LIN {X 0.182,Y -641.756,Z 1201.615,A 0.000,B 0.000,C 90.000,E1 146.755} C_DIS
LIN {X 0.071,Y -644.719,Z 1201.609,A 0.000,B 0.000,C 90.000,E1 145.515} C_DIS
LIN {X -0.049,Y -646.870,Z 1201.603,A 0.000,B 0.000,C 90.000,E1 144.529} C_DIS
LIN {X -0.142,Y -649.015,Z 1201.597,A 0.000,B 0.000,C 90.000,E1 143.543} C_DIS
LIN {X -0.312,Y -652.420,Z 1201.588,A 0.000,B 0.000,C 90.000,E1 141.823} C_DIS
LIN {X 0.039,Y -655.366,Z 1201.580,A 0.000,B 0.000,C 90.000,E1 140.312} C_DIS
LIN {X -0.108,Y -657.902,Z 1201.573,A 0.000,B 0.000,C 90.000,E1 139.094} C_DIS
LIN {X -0.258,Y -661.617,Z 1201.563,A 0.000,B 0.000,C 90.000,E1 137.391} C_DIS
LIN {X 0.141,Y -664.717,Z 1201.555,A 0.000,B 0.000,C 90.000,E1 135.891} C_DIS
LIN {X 0.142,Y -669.639,Z 1201.543,A 0.000,B 0.000,C 90.000,E1 133.704} C_DIS
LIN {X -0.248,Y -673.208,Z 1201.535,A 0.000,B 0.000,C 90.000,E1 132.285} C_DIS
LIN {X 0.461,Y -677.267,Z 1201.526,A 0.000,B 0.000,C 90.000,E1 130.539} C_DIS
LIN {X 0.246,Y -680.325,Z 1201.519,A 0.000,B 0.000,C 90.000,E1 129.358} C_DIS
LIN {X 0.111,Y -683.795,Z 1201.511,A 0.000,B 0.000,C 90.000,E1 127.935} C_DIS
LIN {X -0.220,Y -687.997,Z 1201.502,A 0.000,B 0.000,C 90.000,E1 126.297} C_DIS
LIN {X 0.230,Y -690.319,Z 1201.496,A 0.000,B 0.000,C 90.000,E1 125.311} C_DIS
LIN {X -0.359,Y -694.087,Z 1201.487,A 0.000,B 0.000,C 90.000,E1 123.706} C_DIS
LIN {X 0.019,Y -696.726,Z 1201.481,A 0.000,B 0.000,C 90.000,E1 122.498} C_DIS
LIN {X 0.113,Y -699.622,Z 1201.473,A 0.000,B 0.000,C 90.000,E1 121.082} C_DIS
LIN {X -0.018,Y -701.865,Z 1201.466,A 0.000,B 0.000,C 90.000,E1 119.922} C_DIS
LIN {X 0.413,Y -704.276,Z 1201.458,A 0.000,B 0.000,C 90.000,E1 118.487} C_DIS
LIN {X -0.305,Y -705.247,Z 1201.455,A 0.000,B 0.000,C 90.000,E1 117.847} C_DIS
LIN {X -0.061,Y -705.997,Z 1201.451,A 0.000,B 0.000,C 90.000,E1 117.129} C_DIS
LIN {X 0.185,Y -706.505,Z 1201.447,A 0.000,B 0.000,C 90.000,E1 116.411} C_DIS
LIN {X 0.121,Y -706.839,Z 1201.443,A 0.000,B 0.000,C 90.000,E1 115.720} C_DIS
LIN {X 0.359,Y -706.602,Z 1201.438,A 0.000,B 0.000,C 90.000,E1 114.771} C_DIS
LIN {X -0.285,Y -706.509,Z 1201.437,A 0.000,B 0.000,C 90.000,E1 114.591} C_DIS
LIN {X 0.301,Y -705.614,Z 1201.434,A 0.000,B 0.000,C 90.000,E1 114.079} C_DIS
LIN {X -0.341,Y -705.054,Z 1201.433,A 0.000,B 0.000,C 90.000,E1 113.898} C_DIS
LIN {X 0.370,Y -702.345,Z 1201.429,A 0.000,B 0.000,C 90.000,E1 113.259} C_DIS
LIN {X -0.412,Y -701.469,Z 1201.429,A 0.000,B 0.000,C 90.000,E1 113.206} C_DIS
LIN {X -0.138,Y -698.737,Z 1201.427,A 0.000,B 0.000,C 90.000,E1 112.950} C_DIS
LIN {X 0.063,Y -694.933,Z 1201.426,A 0.000,B 0.000,C 90.000,E1 112.642} C_DIS
LIN {X 0.345,Y -692.825,Z 1201.425,A 0.000,B 0.000,C 90.000,E1 112.514} C_DIS
LIN {X -0.004,Y -686.099,Z 1201.424,A 0.000,B 0.000,C 90.000,E1 112.333} C_DIS
LIN {X -0.355,Y -684.266,Z 1201.424,A 0.000,B 0.000,C 90.000,E1 112.333} C_DIS
LIN {X 0.013,Y -677.402,Z 1201.424,A 0.000,B 0.000,C 90.000,E1 112.280} C_DIS
LIN {X -0.035,Y -608.626,Z 1201.424,A 0.000,B 0.000,C 90.000,E1 112.280} C_DIS
LIN {X -0.207,Y -604.410,Z 1201.422,A 0.000,B 0.000,C 90.000,E1 112.025} C_DIS
LIN {X 0.132,Y -601.624,Z 1201.421,A 0.000,B 0.000,C 90.000,E1 111.791} C_DIS
LIN {X 0.166,Y -587.743,Z 1201.415,A 0.000,B 0.000,C 90.000,E1 110.663} C_DIS
LIN {X -0.026,Y -583.901,Z 1201.413,A 0.000,B 0.000,C 90.000,E1 110.375} C_DIS
LIN {X -0.062,Y -583.880,Z 1201.413,A 0.000,B 0.000,C 90.000,E1 110.375} C_DIS
LIN {X 0.086,Y -583.146,Z 1201.412,A 0.000,B 0.000,C 90.000,E1 110.194} C_DIS
LIN {X 0.080,Y -581.858,Z 1201.411,A 0.000,B 0.000,C 90.000,E1 109.993} C_DIS
LIN {X 0.285,Y -581.582,Z 1201.411,A 0.000,B 0.000,C 90.000,E1 109.939} C_DIS
LIN {X 0.242,Y -581.574,Z 1201.411,A 0.000,B 0.000,C 90.000,E1 109.939} C_DIS
LIN {X -0.205,Y -581.639,Z 1201.409,A 0.000,B 0.000,C 90.000,E1 109.685} C_DIS
LIN {X 0.040,Y -585.854,Z 1201.401,A 0.000,B 0.000,C 90.000,E1 108.181} C_DIS
LIN {X 0.117,Y -587.224,Z 1201.398,A 0.000,B 0.000,C 90.000,E1 107.638} C_DIS
LIN {X -0.118,Y -588.901,Z 1201.394,A 0.000,B 0.000,C 90.000,E1 106.858} C_DIS
LIN {X -0.023,Y -589.809,Z 1201.391,A 0.000,B 0.000,C 90.000,E1 106.315} C_DIS
LIN {X 0.332,Y -590.828,Z 1201.386,A 0.000,B 0.000,C 90.000,E1 105.481} C_DIS
LIN {X 0.281,Y -591.283,Z 1201.383,A 0.000,B 0.000,C 90.000,E1 104.954} C_DIS
LIN {X 0.077,Y -591.263,Z 1201.379,A 0.000,B 0.000,C 90.000,E1 104.175} C_DIS
LIN {X 0.034,Y -591.108,Z 1201.376,A 0.000,B 0.000,C 90.000,E1 103.647} C_DIS
LIN {X -0.008,Y -590.453,Z 1201.373,A 0.000,B 0.000,C 90.000,E1 103.119} C_DIS
LIN {X -0.053,Y -589.382,Z 1201.370,A 0.000,B 0.000,C 90.000,E1 102.591} C_DIS
LIN {X 0.210,Y -588.684,Z 1201.369,A 0.000,B 0.000,C 90.000,E1 102.299} C_DIS
LIN {X 0.154,Y -586.940,Z 1201.365,A 0.000,B 0.000,C 90.000,E1 101.771} C_DIS
LIN {X 0.086,Y -584.803,Z 1201.363,A 0.000,B 0.000,C 90.000,E1 101.243} C_DIS
LIN {X 0.000,Y -582.145,Z 1201.360,A 0.000,B 0.000,C 90.000,E1 100.715} C_DIS
LIN {X 0.011,Y -579.687,Z 1201.357,A 0.000,B 0.000,C 90.000,E1 100.310} C_DIS
LIN {X 0.236,Y -577.742,Z 1201.356,A 0.000,B 0.000,C 90.000,E1 100.018} C_DIS
LIN {X 0.012,Y -573.275,Z 1201.353,A 0.000,B 0.000,C 90.000,E1 99.500} C_DIS
LIN {X -0.067,Y -564.873,Z 1201.348,A 0.000,B 0.000,C 90.000,E1 98.568} C_DIS
LIN {X 0.258,Y -564.024,Z 1201.347,A 0.000,B 0.000,C 90.000,E1 98.398} C_DIS
LIN {X 0.186,Y -562.089,Z 1201.345,A 0.000,B 0.000,C 90.000,E1 97.992} C_DIS
LIN {X 0.023,Y -561.589,Z 1201.344,A 0.000,B 0.000,C 90.000,E1 97.871} C_DIS
LIN {X 0.098,Y -561.138,Z 1201.342,A 0.000,B 0.000,C 90.000,E1 97.587} C_DIS
LIN {X 0.005,Y -560.992,Z 1201.340,A 0.000,B 0.000,C 90.000,E1 97.182} C_DIS
LIN {X -0.074,Y -562.326,Z 1201.326,A 0.000,B 0.000,C 90.000,E1 94.702} C_DIS
LIN {X -0.217,Y -563.102,Z 1201.320,A 0.000,B 0.000,C 90.000,E1 93.612} C_DIS
LIN {X -0.135,Y -564.256,Z 1201.311,A 0.000,B 0.000,C 90.000,E1 91.949} C_DIS
LIN {X 0.084,Y -565.630,Z 1201.300,A 0.000,B 0.000,C 90.000,E1 90.000} C_DIS
LIN {X 0.090,Y -566.626,Z 1201.292,A 0.000,B 0.000,C 90.000,E1 88.625} C_DIS
LIN {X 0.125,Y -567.668,Z 1201.285,A 0.000,B 0.000,C 90.000,E1 87.249} C_DIS
LIN {X -0.234,Y -568.930,Z 1201.276,A 0.000,B 0.000,C 90.000,E1 85.641} C_DIS
LIN {X 0.054,Y -570.177,Z 1201.267,A 0.000,B 0.000,C 90.000,E1 83.970} C_DIS
LIN {X -0.013,Y -571.596,Z 1201.256,A 0.000,B 0.000,C 90.000,E1 82.064} C_DIS
LIN {X 0.204,Y -572.515,Z 1201.248,A 0.000,B 0.000,C 90.000,E1 80.679} C_DIS
LIN {X 0.155,Y -573.575,Z 1201.239,A 0.000,B 0.000,C 90.000,E1 79.050} C_DIS
LIN {X 0.036,Y -574.377,Z 1201.232,A 0.000,B 0.000,C 90.000,E1 77.701} C_DIS
LIN {X -0.083,Y -575.369,Z 1201.221,A 0.000,B 0.000,C 90.000,E1 75.811} C_DIS
LIN {X 0.172,Y -576.215,Z 1201.212,A 0.000,B 0.000,C 90.000,E1 74.157} C_DIS
LIN {X 0.039,Y -577.061,Z 1201.203,A 0.000,B 0.000,C 90.000,E1 72.543} C_DIS
LIN {X -0.279,Y -577.839,Z 1201.196,A 0.000,B 0.000,C 90.000,E1 71.221} C_DIS
LIN {X 0.010,Y -579.305,Z 1201.184,A 0.000,B 0.000,C 90.000,E1 69.028} C_DIS
LIN {X 0.007,Y -581.079,Z 1201.172,A 0.000,B 0.000,C 90.000,E1 66.869} C_DIS
LIN {X 0.250,Y -582.664,Z 1201.163,A 0.000,B 0.000,C 90.000,E1 65.229} C_DIS
LIN {X -0.246,Y -584.659,Z 1201.151,A 0.000,B 0.000,C 90.000,E1 63.127} C_DIS
LIN {X -0.069,Y -586.047,Z 1201.143,A 0.000,B 0.000,C 90.000,E1 61.769} C_DIS
LIN {X 0.298,Y -587.638,Z 1201.134,A 0.000,B 0.000,C 90.000,E1 60.127} C_DIS
LIN {X 0.000,Y -588.858,Z 1201.127,A 0.000,B 0.000,C 90.000,E1 58.820} C_DIS
LIN {X -0.088,Y -590.384,Z 1201.116,A 0.000,B 0.000,C 90.000,E1 56.962} C_DIS
LIN {X 0.279,Y -591.405,Z 1201.109,A 0.000,B 0.000,C 90.000,E1 55.595} C_DIS
LIN {X -0.099,Y -592.618,Z 1201.100,A 0.000,B 0.000,C 90.000,E1 54.036} C_DIS
LIN {X 0.199,Y -593.205,Z 1201.096,A 0.000,B 0.000,C 90.000,E1 53.210} C_DIS
LIN {X -0.012,Y -594.163,Z 1201.088,A 0.000,B 0.000,C 90.000,E1 51.904} C_DIS
LIN {X 0.010,Y -595.129,Z 1201.080,A 0.000,B 0.000,C 90.000,E1 50.312} C_DIS
LIN {X -0.022,Y -595.694,Z 1201.074,A 0.000,B 0.000,C 90.000,E1 49.256} C_DIS
LIN {X 0.124,Y -596.126,Z 1201.066,A 0.000,B 0.000,C 90.000,E1 47.919} C_DIS
LIN {X -0.120,Y -596.431,Z 1201.059,A 0.000,B 0.000,C 90.000,E1 46.620} C_DIS
LIN {X 0.040,Y -596.598,Z 1201.052,A 0.000,B 0.000,C 90.000,E1 45.283} C_DIS
LIN {X -0.006,Y -596.487,Z 1201.046,A 0.000,B 0.000,C 90.000,E1 44.231} C_DIS
LIN {X -0.244,Y -596.255,Z 1201.041,A 0.000,B 0.000,C 90.000,E1 43.461} C_DIS
LIN {X 0.127,Y -595.462,Z 1201.033,A 0.000,B 0.000,C 90.000,E1 41.838} C_DIS
LIN {X -0.128,Y -594.562,Z 1201.025,A 0.000,B 0.000,C 90.000,E1 40.539} C_DIS
LIN {X 0.051,Y -593.454,Z 1201.018,A 0.000,B 0.000,C 90.000,E1 39.197} C_DIS
LIN {X -0.011,Y -592.323,Z 1201.012,A 0.000,B 0.000,C 90.000,E1 38.141} C_DIS
LIN {X 0.010,Y -591.087,Z 1201.006,A 0.000,B 0.000,C 90.000,E1 37.076} C_DIS
LIN {X 0.019,Y -589.596,Z 1201.000,A 0.000,B 0.000,C 90.000,E1 36.011} C_DIS
LIN {X 0.085,Y -588.745,Z 1200.997,A 0.000,B 0.000,C 90.000,E1 35.471} C_DIS
LIN {X 0.254,Y -586.123,Z 1200.990,A 0.000,B 0.000,C 90.000,E1 34.119} C_DIS
LIN {X -0.144,Y -583.324,Z 1200.984,A 0.000,B 0.000,C 90.000,E1 33.086} C_DIS
LIN {X 0.057,Y -580.946,Z 1200.979,A 0.000,B 0.000,C 90.000,E1 32.260} C_DIS
LIN {X 0.072,Y -579.148,Z 1200.976,A 0.000,B 0.000,C 90.000,E1 31.720} C_DIS
LIN {X -0.234,Y -575.010,Z 1200.970,A 0.000,B 0.000,C 90.000,E1 30.669} C_DIS
LIN {X 0.077,Y -571.486,Z 1200.966,A 0.000,B 0.000,C 90.000,E1 29.823} C_DIS
LIN {X 0.036,Y -566.553,Z 1200.960,A 0.000,B 0.000,C 90.000,E1 28.871} C_DIS
LIN {X 0.074,Y -562.813,Z 1200.957,A 0.000,B 0.000,C 90.000,E1 28.180} C_DIS
LIN {X 0.141,Y -556.991,Z 1200.951,A 0.000,B 0.000,C 90.000,E1 27.206} C_DIS
LIN {X 0.243,Y -551.557,Z 1200.947,A 0.000,B 0.000,C 90.000,E1 26.360} C_DIS
LIN {X -0.097,Y -548.695,Z 1200.944,A 0.000,B 0.000,C 90.000,E1 25.976} C_DIS
LIN {X -0.203,Y -543.357,Z 1200.940,A 0.000,B 0.000,C 90.000,E1 25.283} C_DIS
LIN {X 0.007,Y -538.827,Z 1200.937,A 0.000,B 0.000,C 90.000,E1 24.695} C_DIS
LIN {X 0.015,Y -530.380,Z 1200.932,A 0.000,B 0.000,C 90.000,E1 23.695} C_DIS
LIN {X 0.302,Y -523.988,Z 1200.928,A 0.000,B 0.000,C 90.000,E1 22.950} C_DIS
LIN {X 0.036,Y -517.336,Z 1200.924,A 0.000,B 0.000,C 90.000,E1 22.280} C_DIS
LIN {X 0.298,Y -507.842,Z 1200.918,A 0.000,B 0.000,C 90.000,E1 21.280} C_DIS
LIN {X -0.201,Y -496.588,Z 1200.912,A 0.000,B 0.000,C 90.000,E1 20.248} C_DIS
LIN {X 0.125,Y -485.128,Z 1200.906,A 0.000,B 0.000,C 90.000,E1 19.141} C_DIS
LIN {X 0.028,Y -476.168,Z 1200.902,A 0.000,B 0.000,C 90.000,E1 18.362} C_DIS
LIN {X -0.144,Y -464.311,Z 1200.896,A 0.000,B 0.000,C 90.000,E1 17.330} C_DIS
LIN {X -0.099,Y -448.031,Z 1200.888,A 0.000,B 0.000,C 90.000,E1 15.843} C_DIS
LIN {X -0.014,Y -427.765,Z 1200.877,A 0.000,B 0.000,C 90.000,E1 13.828} C_DIS
LIN {X 0.140,Y -415.560,Z 1200.870,A 0.000,B 0.000,C 90.000,E1 12.479} C_DIS
LIN {X 0.104,Y -401.879,Z 1200.860,A 0.000,B 0.000,C 90.000,E1 10.838} C_DIS
LIN {X 0.123,Y -399.353,Z 1200.858,A 0.000,B 0.000,C 90.000,E1 10.489} C_DIS
LIN {X 0.139,Y -395.928,Z 1200.855,A 0.000,B 0.000,C 90.000,E1 9.962} C_DIS
LIN {X 0.034,Y -393.804,Z 1200.853,A 0.000,B 0.000,C 90.000,E1 9.557} C_DIS
LIN {X -0.003,Y -393.795,Z 1200.853,A 0.000,B 0.000,C 90.000,E1 9.557} C_DIS
LIN {X 0.000,Y -393.236,Z 1200.851,A 0.000,B 0.000,C 90.000,E1 9.208} C_DIS
LIN {X -0.037,Y -393.234,Z 1200.851,A 0.000,B 0.000,C 90.000,E1 9.208} C_DIS
LIN {X 0.037,Y -393.785,Z 1200.849,A 0.000,B 0.000,C 90.000,E1 8.859} C_DIS
LIN {X -0.041,Y -395.824,Z 1200.846,A 0.000,B 0.000,C 90.000,E1 8.341} C_DIS
LIN {X 0.144,Y -396.923,Z 1200.845,A 0.000,B 0.000,C 90.000,E1 8.049} C_DIS
LIN {X -0.122,Y -402.735,Z 1200.840,A 0.000,B 0.000,C 90.000,E1 7.296} C_DIS
LIN {X 0.005,Y -405.877,Z 1200.839,A 0.000,B 0.000,C 90.000,E1 6.947} C_DIS
LIN {X 0.017,Y -411.387,Z 1200.836,A 0.000,B 0.000,C 90.000,E1 6.486} C_DIS
LIN {X -0.086,Y -425.657,Z 1200.830,A 0.000,B 0.000,C 90.000,E1 5.391} C_DIS
LIN {X -0.154,Y -441.748,Z 1200.823,A 0.000,B 0.000,C 90.000,E1 4.188} C_DIS
LIN {X 0.085,Y -456.046,Z 1200.817,A 0.000,B 0.000,C 90.000,E1 3.094} C_DIS
LIN {X -0.057,Y -465.616,Z 1200.813,A 0.000,B 0.000,C 90.000,E1 2.407} C_DIS
LIN {X -0.205,Y -474.695,Z 1200.809,A 0.000,B 0.000,C 90.000,E1 1.718} C_DIS
LIN {X 0.098,Y -479.239,Z 1200.807,A 0.000,B 0.000,C 90.000,E1 1.318} C_DIS
LIN {X -0.164,Y -485.056,Z 1200.805,A 0.000,B 0.000,C 90.000,E1 0.859} C_DIS
LIN {X -0.221,Y -490.876,Z 1200.802,A 0.000,B 0.000,C 90.000,E1 0.344} C_DIS
LIN {X -0.012,Y -497.588,Z 1200.798,A 0.000,B 0.000,C 90.000,E1 359.656} C_DIS
LIN {X -0.013,Y -504.065,Z 1200.794,A 0.000,B 0.000,C 90.000,E1 358.969} C_DIS
LIN {X 0.007,Y -511.334,Z 1200.790,A 0.000,B 0.000,C 90.000,E1 358.108} C_DIS
LIN {X -0.163,Y -516.119,Z 1200.786,A 0.000,B 0.000,C 90.000,E1 357.535} C_DIS
LIN {X 0.184,Y -522.568,Z 1200.781,A 0.000,B 0.000,C 90.000,E1 356.617} C_DIS
LIN {X 0.087,Y -526.516,Z 1200.778,A 0.000,B 0.000,C 90.000,E1 356.045} C_DIS
LIN {X -0.227,Y -530.973,Z 1200.774,A 0.000,B 0.000,C 90.000,E1 355.355} C_DIS
LIN {X -0.231,Y -534.312,Z 1200.771,A 0.000,B 0.000,C 90.000,E1 354.780} C_DIS
LIN {X 0.053,Y -537.938,Z 1200.767,A 0.000,B 0.000,C 90.000,E1 354.033} C_DIS
LIN {X 0.166,Y -541.886,Z 1200.762,A 0.000,B 0.000,C 90.000,E1 353.166} C_DIS
LIN {X 0.243,Y -544.317,Z 1200.759,A 0.000,B 0.000,C 90.000,E1 352.591} C_DIS
LIN {X -0.121,Y -547.712,Z 1200.754,A 0.000,B 0.000,C 90.000,E1 351.781} C_DIS
LIN {X 0.178,Y -550.689,Z 1200.750,A 0.000,B 0.000,C 90.000,E1 350.905} C_DIS
LIN {X 0.000,Y -554.167,Z 1200.743,A 0.000,B 0.000,C 90.000,E1 349.803} C_DIS
LIN {X -0.004,Y -558.104,Z 1200.736,A 0.000,B 0.000,C 90.000,E1 348.409} C_DIS
LIN {X -0.131,Y -560.195,Z 1200.731,A 0.000,B 0.000,C 90.000,E1 347.589} C_DIS
LIN {X 0.045,Y -562.828,Z 1200.725,A 0.000,B 0.000,C 90.000,E1 346.464} C_DIS
LIN {X -0.115,Y -565.828,Z 1200.717,A 0.000,B 0.000,C 90.000,E1 345.102} C_DIS
LIN {X -0.228,Y -568.595,Z 1200.710,A 0.000,B 0.000,C 90.000,E1 343.740} C_DIS
LIN {X -0.138,Y -571.129,Z 1200.702,A 0.000,B 0.000,C 90.000,E1 342.362} C_DIS
LIN {X 0.189,Y -572.538,Z 1200.697,A 0.000,B 0.000,C 90.000,E1 341.511} C_DIS
LIN {X 0.167,Y -574.225,Z 1200.691,A 0.000,B 0.000,C 90.000,E1 340.423} C_DIS
LIN {X 0.159,Y -575.636,Z 1200.685,A 0.000,B 0.000,C 90.000,E1 339.337} C_DIS
LIN {X -0.006,Y -576.462,Z 1200.681,A 0.000,B 0.000,C 90.000,E1 338.539} C_DIS
LIN {X -0.321,Y -577.242,Z 1200.675,A 0.000,B 0.000,C 90.000,E1 337.486} C_DIS
LIN {X -0.246,Y -577.486,Z 1200.670,A 0.000,B 0.000,C 90.000,E1 336.666} C_DIS
LIN {X -0.163,Y -577.519,Z 1200.666,A 0.000,B 0.000,C 90.000,E1 335.845} C_DIS
LIN {X -0.077,Y -577.085,Z 1200.661,A 0.000,B 0.000,C 90.000,E1 335.025} C_DIS
LIN {X 0.151,Y -576.688,Z 1200.658,A 0.000,B 0.000,C 90.000,E1 334.460} C_DIS
LIN {X 0.223,Y -575.621,Z 1200.654,A 0.000,B 0.000,C 90.000,E1 333.640} C_DIS
LIN {X -0.233,Y -574.234,Z 1200.649,A 0.000,B 0.000,C 90.000,E1 332.871} C_DIS
LIN {X 0.069,Y -572.429,Z 1200.645,A 0.000,B 0.000,C 90.000,E1 332.025} C_DIS
LIN {X 0.353,Y -570.370,Z 1200.640,A 0.000,B 0.000,C 90.000,E1 331.179} C_DIS
LIN {X 0.012,Y -568.722,Z 1200.637,A 0.000,B 0.000,C 90.000,E1 330.667} C_DIS
LIN {X -0.061,Y -566.883,Z 1200.634,A 0.000,B 0.000,C 90.000,E1 330.127} C_DIS
LIN {X 0.154,Y -563.285,Z 1200.630,A 0.000,B 0.000,C 90.000,E1 329.282} C_DIS
LIN {X -0.058,Y -559.614,Z 1200.626,A 0.000,B 0.000,C 90.000,E1 328.614} C_DIS
LIN {X -0.008,Y -555.289,Z 1200.622,A 0.000,B 0.000,C 90.000,E1 327.916} C_DIS
LIN {X -0.168,Y -551.454,Z 1200.619,A 0.000,B 0.000,C 90.000,E1 327.375} C_DIS
LIN {X 0.015,Y -544.067,Z 1200.613,A 0.000,B 0.000,C 90.000,E1 326.373} C_DIS
LIN {X -0.066,Y -538.317,Z 1200.609,A 0.000,B 0.000,C 90.000,E1 325.674} C_DIS
LIN {X -0.068,Y -526.092,Z 1200.601,A 0.000,B 0.000,C 90.000,E1 324.242} C_DIS
LIN {X 0.158,Y -522.387,Z 1200.599,A 0.000,B 0.000,C 90.000,E1 323.783} C_DIS
LIN {X -0.044,Y -518.272,Z 1200.596,A 0.000,B 0.000,C 90.000,E1 323.256} C_DIS
LIN {X -0.279,Y -515.464,Z 1200.594,A 0.000,B 0.000,C 90.000,E1 322.844} C_DIS
LIN {X -0.203,Y -513.285,Z 1200.591,A 0.000,B 0.000,C 90.000,E1 322.351} C_DIS
LIN {X -0.040,Y -511.726,Z 1200.588,A 0.000,B 0.000,C 90.000,E1 321.743} C_DIS
LIN {X -0.288,Y -511.005,Z 1200.583,A 0.000,B 0.000,C 90.000,E1 320.884} C_DIS
LIN {X 0.063,Y -512.491,Z 1200.564,A 0.000,B 0.000,C 90.000,E1 317.595} C_DIS
LIN {X -0.076,Y -513.345,Z 1200.556,A 0.000,B 0.000,C 90.000,E1 316.134} C_DIS
LIN {X -0.220,Y -514.213,Z 1200.548,A 0.000,B 0.000,C 90.000,E1 314.676} C_DIS
LIN {X 0.022,Y -515.029,Z 1200.540,A 0.000,B 0.000,C 90.000,E1 313.176} C_DIS
LIN {X -0.261,Y -516.176,Z 1200.528,A 0.000,B 0.000,C 90.000,E1 311.148} C_DIS
LIN {X 0.058,Y -517.085,Z 1200.520,A 0.000,B 0.000,C 90.000,E1 309.644} C_DIS
LIN {X 0.126,Y -517.776,Z 1200.514,A 0.000,B 0.000,C 90.000,E1 308.463} C_DIS
LIN {X -0.115,Y -518.301,Z 1200.507,A 0.000,B 0.000,C 90.000,E1 307.317} C_DIS
LIN {X 0.207,Y -519.233,Z 1200.496,A 0.000,B 0.000,C 90.000,E1 305.231} C_DIS
LIN {X -0.001,Y -520.123,Z 1200.486,A 0.000,B 0.000,C 90.000,E1 303.499} C_DIS
LIN {X -0.081,Y -520.651,Z 1200.480,A 0.000,B 0.000,C 90.000,E1 302.339} C_DIS
LIN {X -0.043,Y -521.158,Z 1200.472,A 0.000,B 0.000,C 90.000,E1 300.875} C_DIS
LIN {X -0.051,Y -521.412,Z 1200.467,A 0.000,B 0.000,C 90.000,E1 300.001} C_DIS
LIN {X 0.129,Y -521.650,Z 1200.457,A 0.000,B 0.000,C 90.000,E1 298.231} C_DIS
LIN {X -0.077,Y -521.844,Z 1200.449,A 0.000,B 0.000,C 90.000,E1 296.796} C_DIS
LIN {X -0.053,Y -521.959,Z 1200.441,A 0.000,B 0.000,C 90.000,E1 295.335} C_DIS
LIN {X -0.241,Y -521.931,Z 1200.433,A 0.000,B 0.000,C 90.000,E1 293.898} C_DIS
LIN {X -0.114,Y -521.975,Z 1200.421,A 0.000,B 0.000,C 90.000,E1 291.844} C_DIS
LIN {X -0.008,Y -521.910,Z 1200.413,A 0.000,B 0.000,C 90.000,E1 290.375} C_DIS
LIN {X -0.058,Y -521.600,Z 1200.407,A 0.000,B 0.000,C 90.000,E1 289.214} C_DIS
LIN {X -0.267,Y -521.395,Z 1200.402,A 0.000,B 0.000,C 90.000,E1 288.362} C_DIS
LIN {X 0.143,Y -520.561,Z 1200.394,A 0.000,B 0.000,C 90.000,E1 286.858} C_DIS
LIN {X -0.113,Y -519.795,Z 1200.386,A 0.000,B 0.000,C 90.000,E1 285.426} C_DIS
LIN {X 0.094,Y -518.292,Z 1200.374,A 0.000,B 0.000,C 90.000,E1 283.355} C_DIS
LIN {X 0.150,Y -517.154,Z 1200.365,A 0.000,B 0.000,C 90.000,E1 281.591} C_DIS
LIN {X 0.004,Y -516.472,Z 1200.358,A 0.000,B 0.000,C 90.000,E1 280.433} C_DIS
LIN {X -0.189,Y -515.321,Z 1200.347,A 0.000,B 0.000,C 90.000,E1 278.398} C_DIS
LIN {X 0.132,Y -514.419,Z 1200.338,A 0.000,B 0.000,C 90.000,E1 276.891} C_DIS
LIN {X -0.109,Y -513.750,Z 1200.332,A 0.000,B 0.000,C 90.000,E1 275.739} C_DIS
LIN {X -0.063,Y -512.602,Z 1200.320,A 0.000,B 0.000,C 90.000,E1 273.669} C_DIS
LIN {X -0.171,Y -511.356,Z 1200.307,A 0.000,B 0.000,C 90.000,E1 271.318} C_DIS
LIN {X -0.253,Y -510.356,Z 1200.296,A 0.000,B 0.000,C 90.000,E1 269.255} C_DIS
LIN {X 0.248,Y -509.218,Z 1200.286,A 0.000,B 0.000,C 90.000,E1 267.421} C_DIS
LIN {X -0.204,Y -508.266,Z 1200.278,A 0.000,B 0.000,C 90.000,E1 265.988} C_DIS
LIN {X -0.030,Y -507.342,Z 1200.271,A 0.000,B 0.000,C 90.000,E1 264.780} C_DIS
LIN {X 0.246,Y -506.509,Z 1200.266,A 0.000,B 0.000,C 90.000,E1 263.856} C_DIS
LIN {X 0.276,Y -504.859,Z 1200.256,A 0.000,B 0.000,C 90.000,E1 262.064} C_DIS
LIN {X -0.235,Y -503.362,Z 1200.246,A 0.000,B 0.000,C 90.000,E1 260.330} C_DIS
LIN {X -0.254,Y -501.505,Z 1200.233,A 0.000,B 0.000,C 90.000,E1 257.937} C_DIS
LIN {X 0.069,Y -500.446,Z 1200.226,A 0.000,B 0.000,C 90.000,E1 256.700} C_DIS
LIN {X -0.187,Y -499.281,Z 1200.218,A 0.000,B 0.000,C 90.000,E1 255.227} C_DIS
LIN {X 0.159,Y -496.969,Z 1200.199,A 0.000,B 0.000,C 90.000,E1 251.873} C_DIS
LIN {X 0.165,Y -496.264,Z 1200.194,A 0.000,B 0.000,C 90.000,E1 250.967} C_DIS
LIN {X 0.089,Y -495.155,Z 1200.186,A 0.000,B 0.000,C 90.000,E1 249.464} C_DIS
LIN {X -0.127,Y -493.843,Z 1200.178,A 0.000,B 0.000,C 90.000,E1 247.975} C_DIS
LIN {X 0.091,Y -492.395,Z 1200.169,A 0.000,B 0.000,C 90.000,E1 246.433} C_DIS
LIN {X 0.023,Y -490.882,Z 1200.161,A 0.000,B 0.000,C 90.000,E1 244.921} C_DIS
LIN {X -0.099,Y -489.578,Z 1200.154,A 0.000,B 0.000,C 90.000,E1 243.717} C_DIS
LIN {X 0.216,Y -487.801,Z 1200.146,A 0.000,B 0.000,C 90.000,E1 242.153} C_DIS
LIN {X -0.157,Y -486.324,Z 1200.139,A 0.000,B 0.000,C 90.000,E1 240.973} C_DIS
LIN {X 0.098,Y -484.407,Z 1200.130,A 0.000,B 0.000,C 90.000,E1 239.410} C_DIS
LIN {X -0.083,Y -482.861,Z 1200.123,A 0.000,B 0.000,C 90.000,E1 238.201} C_DIS
LIN {X -0.005,Y -480.548,Z 1200.113,A 0.000,B 0.000,C 90.000,E1 236.342} C_DIS
LIN {X 0.020,Y -478.303,Z 1200.103,A 0.000,B 0.000,C 90.000,E1 234.482} C_DIS
LIN {X -0.103,Y -476.844,Z 1200.096,A 0.000,B 0.000,C 90.000,E1 233.256} C_DIS
LIN {X 0.256,Y -473.859,Z 1200.082,A 0.000,B 0.000,C 90.000,E1 230.723} C_DIS
LIN {X 0.138,Y -472.113,Z 1200.073,A 0.000,B 0.000,C 90.000,E1 229.175} C_DIS
LIN {X 0.100,Y -469.494,Z 1200.061,A 0.000,B 0.000,C 90.000,E1 226.986} C_DIS
LIN {X -0.264,Y -466.893,Z 1200.047,A 0.000,B 0.000,C 90.000,E1 224.514} C_DIS
LIN {X 0.043,Y -464.593,Z 1200.031,A 0.000,B 0.000,C 90.000,E1 221.634} C_DIS
LIN {X 0.023,Y -464.116,Z 1200.001,A 0.000,B 0.000,C 90.000,E1 216.251} C_DIS
LIN {X 0.113,Y -464.624,Z 1199.987,A 0.000,B 0.000,C 90.000,E1 213.706} C_DIS
LIN {X 0.039,Y -467.527,Z 1199.966,A 0.000,B 0.000,C 90.000,E1 209.922} C_DIS
LIN {X 0.198,Y -470.208,Z 1199.952,A 0.000,B 0.000,C 90.000,E1 207.385} C_DIS
LIN {X -0.170,Y -471.373,Z 1199.947,A 0.000,B 0.000,C 90.000,E1 206.488} C_DIS
LIN {X -0.002,Y -476.354,Z 1199.926,A 0.000,B 0.000,C 90.000,E1 202.717} C_DIS
LIN {X -0.141,Y -482.595,Z 1199.907,A 0.000,B 0.000,C 90.000,E1 199.322} C_DIS
LIN {X 0.266,Y -490.733,Z 1199.889,A 0.000,B 0.000,C 90.000,E1 195.898} C_DIS
LIN {X 0.198,Y -498.346,Z 1199.873,A 0.000,B 0.000,C 90.000,E1 193.175} C_DIS
LIN {X 0.176,Y -504.704,Z 1199.862,A 0.000,B 0.000,C 90.000,E1 191.074} C_DIS
LIN {X -0.178,Y -511.313,Z 1199.850,A 0.000,B 0.000,C 90.000,E1 189.029} C_DIS
LIN {X 0.017,Y -516.244,Z 1199.842,A 0.000,B 0.000,C 90.000,E1 187.530} C_DIS
LIN {X -0.200,Y -521.021,Z 1199.834,A 0.000,B 0.000,C 90.000,E1 186.087} C_DIS
LIN {X 0.140,Y -526.621,Z 1199.824,A 0.000,B 0.000,C 90.000,E1 184.302} C_DIS
LIN {X 0.052,Y -531.308,Z 1199.816,A 0.000,B 0.000,C 90.000,E1 182.865} C_DIS
LIN {X 0.021,Y -537.813,Z 1199.805,A 0.000,B 0.000,C 90.000,E1 180.859} C_DIS
LIN {X 0.147,Y -544.305,Z 1199.794,A 0.000,B 0.000,C 90.000,E1 178.854} C_DIS
LIN {X -0.105,Y -550.622,Z 1199.783,A 0.000,B 0.000,C 90.000,E1 176.906} C_DIS
LIN {X 0.184,Y -554.114,Z 1199.777,A 0.000,B 0.000,C 90.000,E1 175.755} C_DIS
LIN {X 0.121,Y -559.305,Z 1199.767,A 0.000,B 0.000,C 90.000,E1 174.090} C_DIS
LIN {X 0.131,Y -563.503,Z 1199.760,A 0.000,B 0.000,C 90.000,E1 172.704} C_DIS
LIN {X 0.130,Y -566.846,Z 1199.753,A 0.000,B 0.000,C 90.000,E1 171.602} C_DIS
LIN {X -0.293,Y -570.991,Z 1199.746,A 0.000,B 0.000,C 90.000,E1 170.274} C_DIS
LIN {X 0.111,Y -575.081,Z 1199.738,A 0.000,B 0.000,C 90.000,E1 168.870} C_DIS
LIN {X 0.035,Y -579.170,Z 1199.731,A 0.000,B 0.000,C 90.000,E1 167.521} C_DIS
LIN {X 0.260,Y -584.149,Z 1199.722,A 0.000,B 0.000,C 90.000,E1 165.880} C_DIS
LIN {X 0.153,Y -589.123,Z 1199.713,A 0.000,B 0.000,C 90.000,E1 164.283} C_DIS
LIN {X -0.126,Y -595.766,Z 1199.701,A 0.000,B 0.000,C 90.000,E1 162.181} C_DIS
LIN {X 0.182,Y -599.202,Z 1199.695,A 0.000,B 0.000,C 90.000,E1 161.094} C_DIS
LIN {X 0.087,Y -605.116,Z 1199.685,A 0.000,B 0.000,C 90.000,E1 159.263} C_DIS
LIN {X 0.122,Y -611.115,Z 1199.675,A 0.000,B 0.000,C 90.000,E1 157.433} C_DIS
LIN {X -0.035,Y -614.474,Z 1199.669,A 0.000,B 0.000,C 90.000,E1 156.410} C_DIS
LIN {X 0.144,Y -619.408,Z 1199.660,A 0.000,B 0.000,C 90.000,E1 154.845} C_DIS
LIN {X -0.154,Y -623.291,Z 1199.653,A 0.000,B 0.000,C 90.000,E1 153.589} C_DIS
LIN {X 0.184,Y -627.832,Z 1199.645,A 0.000,B 0.000,C 90.000,E1 152.025} C_DIS
LIN {X -0.262,Y -631.424,Z 1199.638,A 0.000,B 0.000,C 90.000,E1 150.795} C_DIS
LIN {X 0.014,Y -635.650,Z 1199.629,A 0.000,B 0.000,C 90.000,E1 149.253} C_DIS
LIN {X 0.003,Y -638.963,Z 1199.622,A 0.000,B 0.000,C 90.000,E1 147.995} C_DIS
LIN {X -0.159,Y -642.053,Z 1199.615,A 0.000,B 0.000,C 90.000,E1 146.755} C_DIS
LIN {X 0.265,Y -644.954,Z 1199.608,A 0.000,B 0.000,C 90.000,E1 145.468} C_DIS
LIN {X -0.281,Y -646.610,Z 1199.604,A 0.000,B 0.000,C 90.000,E1 144.769} C_DIS
LIN {X 0.047,Y -649.181,Z 1199.597,A 0.000,B 0.000,C 90.000,E1 143.497} C_DIS
LIN {X -0.174,Y -652.034,Z 1199.589,A 0.000,B 0.000,C 90.000,E1 142.029} C_DIS
LIN {X 0.177,Y -654.983,Z 1199.581,A 0.000,B 0.000,C 90.000,E1 140.517} C_DIS
LIN {X 0.020,Y -658.487,Z 1199.571,A 0.000,B 0.000,C 90.000,E1 138.809} C_DIS
LIN {X 0.345,Y -661.707,Z 1199.563,A 0.000,B 0.000,C 90.000,E1 137.310} C_DIS
LIN {X -0.191,Y -664.792,Z 1199.555,A 0.000,B 0.000,C 90.000,E1 135.891} C_DIS
LIN {X -0.191,Y -669.708,Z 1199.543,A 0.000,B 0.000,C 90.000,E1 133.704} C_DIS
LIN {X -0.064,Y -673.859,Z 1199.533,A 0.000,B 0.000,C 90.000,E1 132.000} C_DIS
LIN {X -0.236,Y -679.136,Z 1199.521,A 0.000,B 0.000,C 90.000,E1 129.850} C_DIS
LIN {X 0.105,Y -682.106,Z 1199.515,A 0.000,B 0.000,C 90.000,E1 128.624} C_DIS
LIN {X 0.195,Y -686.835,Z 1199.504,A 0.000,B 0.000,C 90.000,E1 126.710} C_DIS
LIN {X -0.336,Y -689.215,Z 1199.499,A 0.000,B 0.000,C 90.000,E1 125.804} C_DIS
LIN {X 0.130,Y -691.418,Z 1199.494,A 0.000,B 0.000,C 90.000,E1 124.818} C_DIS
LIN {X -0.088,Y -694.667,Z 1199.486,A 0.000,B 0.000,C 90.000,E1 123.420} C_DIS
LIN {X 0.055,Y -696.758,Z 1199.480,A 0.000,B 0.000,C 90.000,E1 122.467} C_DIS
LIN {X 0.136,Y -699.649,Z 1199.473,A 0.000,B 0.000,C 90.000,E1 121.052} C_DIS
LIN {X 0.250,Y -701.885,Z 1199.466,A 0.000,B 0.000,C 90.000,E1 119.873} C_DIS
LIN {X -0.209,Y -703.917,Z 1199.460,A 0.000,B 0.000,C 90.000,E1 118.743} C_DIS
LIN {X 0.307,Y -705.246,Z 1199.454,A 0.000,B 0.000,C 90.000,E1 117.769} C_DIS
LIN {X 0.226,Y -705.995,Z 1199.451,A 0.000,B 0.000,C 90.000,E1 117.078} C_DIS
LIN {X -0.156,Y -706.495,Z 1199.447,A 0.000,B 0.000,C 90.000,E1 116.411} C_DIS
LIN {X -0.221,Y -706.823,Z 1199.443,A 0.000,B 0.000,C 90.000,E1 115.720} C_DIS
LIN {X 0.016,Y -706.590,Z 1199.438,A 0.000,B 0.000,C 90.000,E1 114.771} C_DIS
LIN {X 0.309,Y -706.485,Z 1199.436,A 0.000,B 0.000,C 90.000,E1 114.515} C_DIS
LIN {X -0.041,Y -705.557,Z 1199.434,A 0.000,B 0.000,C 90.000,E1 114.079} C_DIS
LIN {X 0.247,Y -704.940,Z 1199.432,A 0.000,B 0.000,C 90.000,E1 113.823} C_DIS
LIN {X -0.110,Y -702.772,Z 1199.430,A 0.000,B 0.000,C 90.000,E1 113.387} C_DIS
LIN {X 0.029,Y -702.131,Z 1199.429,A 0.000,B 0.000,C 90.000,E1 113.259} C_DIS
LIN {X 0.168,Y -701.165,Z 1199.429,A 0.000,B 0.000,C 90.000,E1 113.131} C_DIS
LIN {X -0.246,Y -697.104,Z 1199.427,A 0.000,B 0.000,C 90.000,E1 112.823} C_DIS
LIN {X -0.015,Y -695.691,Z 1199.426,A 0.000,B 0.000,C 90.000,E1 112.695} C_DIS
LIN {X 0.010,Y -694.055,Z 1199.426,A 0.000,B 0.000,C 90.000,E1 112.589} C_DIS
LIN {X 0.300,Y -691.220,Z 1199.425,A 0.000,B 0.000,C 90.000,E1 112.461} C_DIS
LIN {X -0.101,Y -685.841,Z 1199.424,A 0.000,B 0.000,C 90.000,E1 112.333} C_DIS
LIN {X 0.238,Y -684.133,Z 1199.424,A 0.000,B 0.000,C 90.000,E1 112.280} C_DIS
LIN {X -0.029,Y -677.014,Z 1199.424,A 0.000,B 0.000,C 90.000,E1 112.280} C_DIS
LIN {X -0.074,Y -608.255,Z 1199.424,A 0.000,B 0.000,C 90.000,E1 112.280} C_DIS
LIN {X -0.076,Y -602.461,Z 1199.422,A 0.000,B 0.000,C 90.000,E1 111.897} C_DIS
LIN {X -0.078,Y -589.632,Z 1199.416,A 0.000,B 0.000,C 90.000,E1 110.865} C_DIS
LIN {X -0.148,Y -582.456,Z 1199.413,A 0.000,B 0.000,C 90.000,E1 110.301} C_DIS
LIN {X -0.037,Y -580.309,Z 1199.411,A 0.000,B 0.000,C 90.000,E1 110.066} C_DIS
LIN {X -0.212,Y -578.361,Z 1199.411,A 0.000,B 0.000,C 90.000,E1 109.939} C_DIS
LIN {X -0.155,Y -578.138,Z 1199.410,A 0.000,B 0.000,C 90.000,E1 109.885} C_DIS
LIN {X -0.063,Y -578.010,Z 1199.410,A 0.000,B 0.000,C 90.000,E1 109.812} C_DIS
LIN {X -0.201,Y -578.024,Z 1199.410,A 0.000,B 0.000,C 90.000,E1 109.758} C_DIS
LIN {X 0.124,Y -580.593,Z 1199.404,A 0.000,B 0.000,C 90.000,E1 108.779} C_DIS
LIN {X 0.162,Y -582.191,Z 1199.401,A 0.000,B 0.000,C 90.000,E1 108.236} C_DIS
LIN {X 0.212,Y -583.577,Z 1199.398,A 0.000,B 0.000,C 90.000,E1 107.692} C_DIS
LIN {X 0.098,Y -584.748,Z 1199.396,A 0.000,B 0.000,C 90.000,E1 107.166} C_DIS
LIN {X -0.159,Y -586.087,Z 1199.391,A 0.000,B 0.000,C 90.000,E1 106.386} C_DIS
LIN {X -0.083,Y -586.825,Z 1199.388,A 0.000,B 0.000,C 90.000,E1 105.843} C_DIS
LIN {X -0.006,Y -587.248,Z 1199.385,A 0.000,B 0.000,C 90.000,E1 105.300} C_DIS
LIN {X 0.240,Y -587.453,Z 1199.384,A 0.000,B 0.000,C 90.000,E1 105.009} C_DIS
LIN {X 0.102,Y -587.177,Z 1199.378,A 0.000,B 0.000,C 90.000,E1 103.953} C_DIS
LIN {X -0.077,Y -586.967,Z 1199.376,A 0.000,B 0.000,C 90.000,E1 103.703} C_DIS
LIN {X -0.148,Y -586.224,Z 1199.373,A 0.000,B 0.000,C 90.000,E1 103.175} C_DIS
LIN {X -0.222,Y -584.964,Z 1199.370,A 0.000,B 0.000,C 90.000,E1 102.647} C_DIS
LIN {X 0.266,Y -583.196,Z 1199.367,A 0.000,B 0.000,C 90.000,E1 102.063} C_DIS
LIN {X 0.173,Y -581.043,Z 1199.364,A 0.000,B 0.000,C 90.000,E1 101.535} C_DIS
LIN {X -0.164,Y -579.758,Z 1199.363,A 0.000,B 0.000,C 90.000,E1 101.299} C_DIS
LIN {X 0.174,Y -576.867,Z 1199.360,A 0.000,B 0.000,C 90.000,E1 100.725} C_DIS
LIN {X 0.033,Y -572.775,Z 1199.357,A 0.000,B 0.000,C 90.000,E1 100.197} C_DIS
LIN {X 0.044,Y -565.746,Z 1199.352,A 0.000,B 0.000,C 90.000,E1 99.378} C_DIS
LIN {X -0.194,Y -564.717,Z 1199.351,A 0.000,B 0.000,C 90.000,E1 99.265} C_DIS
LIN {X 0.207,Y -562.437,Z 1199.349,A 0.000,B 0.000,C 90.000,E1 98.746} C_DIS
LIN {X 0.052,Y -561.620,Z 1199.348,A 0.000,B 0.000,C 90.000,E1 98.624} C_DIS
LIN {X 0.243,Y -560.850,Z 1199.347,A 0.000,B 0.000,C 90.000,E1 98.398} C_DIS
LIN {X 0.075,Y -560.636,Z 1199.346,A 0.000,B 0.000,C 90.000,E1 98.276} C_DIS
LIN {X -0.268,Y -560.532,Z 1199.343,A 0.000,B 0.000,C 90.000,E1 97.757} C_DIS
LIN {X -0.137,Y -562.268,Z 1199.326,A 0.000,B 0.000,C 90.000,E1 94.702} C_DIS
LIN {X -0.183,Y -563.190,Z 1199.318,A 0.000,B 0.000,C 90.000,E1 93.326} C_DIS
LIN {X -0.077,Y -564.360,Z 1199.309,A 0.000,B 0.000,C 90.000,E1 91.661} C_DIS
LIN {X -0.096,Y -565.367,Z 1199.302,A 0.000,B 0.000,C 90.000,E1 90.286} C_DIS
LIN {X -0.094,Y -566.376,Z 1199.294,A 0.000,B 0.000,C 90.000,E1 88.912} C_DIS
LIN {X 0.171,Y -567.792,Z 1199.283,A 0.000,B 0.000,C 90.000,E1 86.963} C_DIS
LIN {X -0.190,Y -569.050,Z 1199.274,A 0.000,B 0.000,C 90.000,E1 85.355} C_DIS
LIN {X -0.021,Y -570.069,Z 1199.266,A 0.000,B 0.000,C 90.000,E1 83.970} C_DIS
LIN {X -0.089,Y -571.478,Z 1199.256,A 0.000,B 0.000,C 90.000,E1 82.064} C_DIS
LIN {X 0.126,Y -572.381,Z 1199.248,A 0.000,B 0.000,C 90.000,E1 80.679} C_DIS
LIN {X 0.074,Y -573.438,Z 1199.239,A 0.000,B 0.000,C 90.000,E1 79.050} C_DIS
LIN {X -0.048,Y -574.239,Z 1199.232,A 0.000,B 0.000,C 90.000,E1 77.701} C_DIS
LIN {X 0.045,Y -575.065,Z 1199.223,A 0.000,B 0.000,C 90.000,E1 76.061} C_DIS
LIN {X -0.120,Y -575.935,Z 1199.214,A 0.000,B 0.000,C 90.000,E1 74.448} C_DIS
LIN {X -0.055,Y -576.899,Z 1199.203,A 0.000,B 0.000,C 90.000,E1 72.543} C_DIS
LIN {X 0.000,Y -577.846,Z 1199.194,A 0.000,B 0.000,C 90.000,E1 70.913} C_DIS
LIN {X -0.092,Y -579.162,Z 1199.183,A 0.000,B 0.000,C 90.000,E1 69.028} C_DIS
LIN {X -0.100,Y -580.939,Z 1199.172,A 0.000,B 0.000,C 90.000,E1 66.869} C_DIS
LIN {X 0.274,Y -582.270,Z 1199.164,A 0.000,B 0.000,C 90.000,E1 65.485} C_DIS
LIN {X -0.234,Y -584.299,Z 1199.152,A 0.000,B 0.000,C 90.000,E1 63.384} C_DIS
LIN {X -0.184,Y -585.928,Z 1199.143,A 0.000,B 0.000,C 90.000,E1 61.769} C_DIS
LIN {X 0.181,Y -587.518,Z 1199.134,A 0.000,B 0.000,C 90.000,E1 60.127} C_DIS
LIN {X 0.067,Y -588.914,Z 1199.125,A 0.000,B 0.000,C 90.000,E1 58.535} C_DIS
LIN {X 0.283,Y -590.237,Z 1199.116,A 0.000,B 0.000,C 90.000,E1 56.914} C_DIS
LIN {X 0.024,Y -591.441,Z 1199.108,A 0.000,B 0.000,C 90.000,E1 55.341} C_DIS
LIN {X -0.150,Y -592.861,Z 1199.097,A 0.000,B 0.000,C 90.000,E1 53.497} C_DIS
LIN {X -0.149,Y -593.974,Z 1199.088,A 0.000,B 0.000,C 90.000,E1 51.904} C_DIS
LIN {X 0.029,Y -594.771,Z 1199.081,A 0.000,B 0.000,C 90.000,E1 50.561} C_DIS
LIN {X 0.224,Y -595.504,Z 1199.074,A 0.000,B 0.000,C 90.000,E1 49.218} C_DIS
LIN {X -0.023,Y -595.942,Z 1199.066,A 0.000,B 0.000,C 90.000,E1 47.919} C_DIS
LIN {X -0.269,Y -596.235,Z 1199.059,A 0.000,B 0.000,C 90.000,E1 46.620} C_DIS
LIN {X -0.316,Y -596.361,Z 1199.053,A 0.000,B 0.000,C 90.000,E1 45.567} C_DIS
LIN {X 0.061,Y -596.303,Z 1199.047,A 0.000,B 0.000,C 90.000,E1 44.474} C_DIS
LIN {X 0.030,Y -595.993,Z 1199.041,A 0.000,B 0.000,C 90.000,E1 43.419} C_DIS
LIN {X 0.190,Y -595.364,Z 1199.034,A 0.000,B 0.000,C 90.000,E1 42.081} C_DIS
LIN {X -0.064,Y -594.447,Z 1199.027,A 0.000,B 0.000,C 90.000,E1 40.782} C_DIS
LIN {X -0.099,Y -593.627,Z 1199.021,A 0.000,B 0.000,C 90.000,E1 39.725} C_DIS
LIN {X -0.151,Y -592.633,Z 1199.015,A 0.000,B 0.000,C 90.000,E1 38.669} C_DIS
LIN {X 0.089,Y -591.077,Z 1199.007,A 0.000,B 0.000,C 90.000,E1 37.317} C_DIS
LIN {X 0.104,Y -589.632,Z 1199.001,A 0.000,B 0.000,C 90.000,E1 36.251} C_DIS
LIN {X 0.239,Y -588.359,Z 1198.997,A 0.000,B 0.000,C 90.000,E1 35.438} C_DIS
LIN {X -0.130,Y -586.293,Z 1198.991,A 0.000,B 0.000,C 90.000,E1 34.405} C_DIS
LIN {X -0.078,Y -585.008,Z 1198.988,A 0.000,B 0.000,C 90.000,E1 33.865} C_DIS
LIN {X 0.147,Y -582.884,Z 1198.984,A 0.000,B 0.000,C 90.000,E1 33.038} C_DIS
LIN {X -0.145,Y -580.470,Z 1198.979,A 0.000,B 0.000,C 90.000,E1 32.260} C_DIS
LIN {X -0.133,Y -578.658,Z 1198.976,A 0.000,B 0.000,C 90.000,E1 31.720} C_DIS
LIN {X 0.344,Y -574.472,Z 1198.970,A 0.000,B 0.000,C 90.000,E1 30.590} C_DIS
LIN {X 0.229,Y -571.511,Z 1198.966,A 0.000,B 0.000,C 90.000,E1 29.922} C_DIS
LIN {X -0.007,Y -567.354,Z 1198.962,A 0.000,B 0.000,C 90.000,E1 29.127} C_DIS
LIN {X -0.059,Y -562.930,Z 1198.957,A 0.000,B 0.000,C 90.000,E1 28.309} C_DIS
LIN {X 0.114,Y -558.009,Z 1198.953,A 0.000,B 0.000,C 90.000,E1 27.462} C_DIS
LIN {X -0.156,Y -553.613,Z 1198.949,A 0.000,B 0.000,C 90.000,E1 26.796} C_DIS
LIN {X -0.222,Y -548.926,Z 1198.945,A 0.000,B 0.000,C 90.000,E1 26.104} C_DIS
LIN {X -0.088,Y -543.693,Z 1198.941,A 0.000,B 0.000,C 90.000,E1 25.387} C_DIS
LIN {X -0.108,Y -539.202,Z 1198.938,A 0.000,B 0.000,C 90.000,E1 24.823} C_DIS
LIN {X -0.002,Y -530.906,Z 1198.932,A 0.000,B 0.000,C 90.000,E1 23.823} C_DIS
LIN {X -0.139,Y -524.588,Z 1198.928,A 0.000,B 0.000,C 90.000,E1 23.131} C_DIS
LIN {X 0.161,Y -518.083,Z 1198.925,A 0.000,B 0.000,C 90.000,E1 22.408} C_DIS
LIN {X -0.082,Y -508.576,Z 1198.919,A 0.000,B 0.000,C 90.000,E1 21.461} C_DIS
LIN {X -0.212,Y -501.560,Z 1198.915,A 0.000,B 0.000,C 90.000,E1 20.791} C_DIS
LIN {X 0.184,Y -494.446,Z 1198.912,A 0.000,B 0.000,C 90.000,E1 20.066} C_DIS
LIN {X 0.124,Y -484.372,Z 1198.906,A 0.000,B 0.000,C 90.000,E1 19.141} C_DIS
LIN {X 0.139,Y -475.603,Z 1198.902,A 0.000,B 0.000,C 90.000,E1 18.362} C_DIS
LIN {X 0.007,Y -465.222,Z 1198.897,A 0.000,B 0.000,C 90.000,E1 17.457} C_DIS
LIN {X -0.104,Y -446.020,Z 1198.887,A 0.000,B 0.000,C 90.000,E1 15.717} C_DIS
LIN {X -0.142,Y -425.764,Z 1198.876,A 0.000,B 0.000,C 90.000,E1 13.703} C_DIS
LIN {X 0.096,Y -413.426,Z 1198.868,A 0.000,B 0.000,C 90.000,E1 12.299} C_DIS
LIN {X 0.157,Y -401.547,Z 1198.860,A 0.000,B 0.000,C 90.000,E1 10.838} C_DIS
LIN {X -0.119,Y -396.824,Z 1198.857,A 0.000,B 0.000,C 90.000,E1 10.197} C_DIS
LIN {X -0.093,Y -395.699,Z 1198.856,A 0.000,B 0.000,C 90.000,E1 10.018} C_DIS
LIN {X 0.124,Y -393.674,Z 1198.853,A 0.000,B 0.000,C 90.000,E1 9.557} C_DIS
LIN {X 0.051,Y -393.216,Z 1198.851,A 0.000,B 0.000,C 90.000,E1 9.208} C_DIS
LIN {X 0.013,Y -393.208,Z 1198.851,A 0.000,B 0.000,C 90.000,E1 9.208} C_DIS
LIN {X -0.187,Y -393.827,Z 1198.849,A 0.000,B 0.000,C 90.000,E1 8.916} C_DIS
LIN {X 0.152,Y -394.377,Z 1198.848,A 0.000,B 0.000,C 90.000,E1 8.690} C_DIS
LIN {X -0.091,Y -396.919,Z 1198.845,A 0.000,B 0.000,C 90.000,E1 8.106} C_DIS
LIN {X 0.038,Y -402.297,Z 1198.841,A 0.000,B 0.000,C 90.000,E1 7.296} C_DIS
LIN {X -0.149,Y -407.003,Z 1198.838,A 0.000,B 0.000,C 90.000,E1 6.834} C_DIS
LIN {X -0.031,Y -425.171,Z 1198.830,A 0.000,B 0.000,C 90.000,E1 5.391} C_DIS
LIN {X 0.012,Y -437.971,Z 1198.825,A 0.000,B 0.000,C 90.000,E1 4.416} C_DIS
LIN {X -0.151,Y -452.178,Z 1198.819,A 0.000,B 0.000,C 90.000,E1 3.383} C_DIS
LIN {X 0.175,Y -466.417,Z 1198.813,A 0.000,B 0.000,C 90.000,E1 2.293} C_DIS
LIN {X 0.107,Y -473.981,Z 1198.810,A 0.000,B 0.000,C 90.000,E1 1.718} C_DIS
LIN {X -0.129,Y -480.026,Z 1198.807,A 0.000,B 0.000,C 90.000,E1 1.260} C_DIS
LIN {X 0.119,Y -484.530,Z 1198.805,A 0.000,B 0.000,C 90.000,E1 0.859} C_DIS
LIN {X 0.125,Y -491.526,Z 1198.801,A 0.000,B 0.000,C 90.000,E1 0.229} C_DIS
LIN {X -0.012,Y -497.556,Z 1198.798,A 0.000,B 0.000,C 90.000,E1 359.656} C_DIS
LIN {X 0.077,Y -504.030,Z 1198.794,A 0.000,B 0.000,C 90.000,E1 358.969} C_DIS
LIN {X -0.100,Y -511.557,Z 1198.789,A 0.000,B 0.000,C 90.000,E1 358.108} C_DIS
LIN {X 0.246,Y -516.376,Z 1198.786,A 0.000,B 0.000,C 90.000,E1 357.478} C_DIS
LIN {X -0.153,Y -521.836,Z 1198.782,A 0.000,B 0.000,C 90.000,E1 356.788} C_DIS
LIN {X -0.017,Y -526.814,Z 1198.778,A 0.000,B 0.000,C 90.000,E1 356.045} C_DIS
LIN {X 0.200,Y -531.270,Z 1198.774,A 0.000,B 0.000,C 90.000,E1 355.298} C_DIS
LIN {X 0.202,Y -534.628,Z 1198.771,A 0.000,B 0.000,C 90.000,E1 354.723} C_DIS
LIN {X -0.045,Y -538.249,Z 1198.767,A 0.000,B 0.000,C 90.000,E1 354.033} C_DIS
LIN {X -0.200,Y -541.622,Z 1198.763,A 0.000,B 0.000,C 90.000,E1 353.337} C_DIS
LIN {X 0.142,Y -543.543,Z 1198.760,A 0.000,B 0.000,C 90.000,E1 352.875} C_DIS
LIN {X -0.210,Y -548.058,Z 1198.754,A 0.000,B 0.000,C 90.000,E1 351.781} C_DIS
LIN {X -0.015,Y -550.074,Z 1198.751,A 0.000,B 0.000,C 90.000,E1 351.197} C_DIS
LIN {X 0.225,Y -552.854,Z 1198.746,A 0.000,B 0.000,C 90.000,E1 350.330} C_DIS
LIN {X 0.044,Y -555.361,Z 1198.742,A 0.000,B 0.000,C 90.000,E1 349.511} C_DIS
LIN {X -0.080,Y -558.478,Z 1198.736,A 0.000,B 0.000,C 90.000,E1 348.409} C_DIS
LIN {X -0.203,Y -560.565,Z 1198.731,A 0.000,B 0.000,C 90.000,E1 347.589} C_DIS
LIN {X -0.021,Y -563.224,Z 1198.725,A 0.000,B 0.000,C 90.000,E1 346.464} C_DIS
LIN {X -0.010,Y -566.831,Z 1198.716,A 0.000,B 0.000,C 90.000,E1 344.810} C_DIS
LIN {X -0.112,Y -569.512,Z 1198.708,A 0.000,B 0.000,C 90.000,E1 343.449} C_DIS
LIN {X 0.163,Y -572.033,Z 1198.700,A 0.000,B 0.000,C 90.000,E1 342.054} C_DIS
LIN {X 0.136,Y -573.849,Z 1198.694,A 0.000,B 0.000,C 90.000,E1 340.967} C_DIS
LIN {X -0.238,Y -575.056,Z 1198.690,A 0.000,B 0.000,C 90.000,E1 340.188} C_DIS
LIN {X -0.036,Y -576.453,Z 1198.684,A 0.000,B 0.000,C 90.000,E1 339.082} C_DIS
LIN {X -0.190,Y -577.202,Z 1198.679,A 0.000,B 0.000,C 90.000,E1 338.284} C_DIS
LIN {X 0.043,Y -577.963,Z 1198.673,A 0.000,B 0.000,C 90.000,E1 337.177} C_DIS
LIN {X 0.125,Y -578.116,Z 1198.669,A 0.000,B 0.000,C 90.000,E1 336.357} C_DIS
LIN {X -0.167,Y -578.134,Z 1198.666,A 0.000,B 0.000,C 90.000,E1 335.845} C_DIS
LIN {X -0.075,Y -577.742,Z 1198.661,A 0.000,B 0.000,C 90.000,E1 335.025} C_DIS
LIN {X 0.013,Y -577.069,Z 1198.657,A 0.000,B 0.000,C 90.000,E1 334.204} C_DIS
LIN {X 0.088,Y -575.884,Z 1198.652,A 0.000,B 0.000,C 90.000,E1 333.384} C_DIS
LIN {X -0.213,Y -574.983,Z 1198.649,A 0.000,B 0.000,C 90.000,E1 332.871} C_DIS
LIN {X -0.060,Y -572.566,Z 1198.643,A 0.000,B 0.000,C 90.000,E1 331.769} C_DIS
LIN {X 0.224,Y -570.433,Z 1198.639,A 0.000,B 0.000,C 90.000,E1 330.923} C_DIS
LIN {X 0.163,Y -568.742,Z 1198.636,A 0.000,B 0.000,C 90.000,E1 330.383} C_DIS
LIN {X -0.012,Y -567.759,Z 1198.634,A 0.000,B 0.000,C 90.000,E1 330.127} C_DIS
LIN {X -0.272,Y -564.244,Z 1198.630,A 0.000,B 0.000,C 90.000,E1 329.331} C_DIS
LIN {X 0.008,Y -560.663,Z 1198.626,A 0.000,B 0.000,C 90.000,E1 328.614} C_DIS
LIN {X 0.067,Y -556.405,Z 1198.622,A 0.000,B 0.000,C 90.000,E1 327.916} C_DIS
LIN {X -0.204,Y -551.548,Z 1198.618,A 0.000,B 0.000,C 90.000,E1 327.248} C_DIS
LIN {X 0.110,Y -545.256,Z 1198.613,A 0.000,B 0.000,C 90.000,E1 326.373} C_DIS
LIN {X 0.038,Y -539.495,Z 1198.609,A 0.000,B 0.000,C 90.000,E1 325.674} C_DIS
LIN {X -0.092,Y -528.516,Z 1198.602,A 0.000,B 0.000,C 90.000,E1 324.402} C_DIS
LIN {X -0.304,Y -522.326,Z 1198.598,A 0.000,B 0.000,C 90.000,E1 323.703} C_DIS
LIN {X 0.168,Y -518.442,Z 1198.595,A 0.000,B 0.000,C 90.000,E1 323.130} C_DIS
LIN {X 0.190,Y -516.111,Z 1198.593,A 0.000,B 0.000,C 90.000,E1 322.763} C_DIS
LIN {X -0.114,Y -513.828,Z 1198.591,A 0.000,B 0.000,C 90.000,E1 322.316} C_DIS
LIN {X 0.100,Y -513.292,Z 1198.590,A 0.000,B 0.000,C 90.000,E1 322.145} C_DIS
LIN {X -0.096,Y -512.097,Z 1198.587,A 0.000,B 0.000,C 90.000,E1 321.698} C_DIS
LIN {X 0.145,Y -511.715,Z 1198.586,A 0.000,B 0.000,C 90.000,E1 321.376} C_DIS
LIN {X -0.021,Y -511.322,Z 1198.582,A 0.000,B 0.000,C 90.000,E1 320.803} C_DIS
LIN {X -0.002,Y -512.840,Z 1198.564,A 0.000,B 0.000,C 90.000,E1 317.553} C_DIS
LIN {X 0.212,Y -513.690,Z 1198.556,A 0.000,B 0.000,C 90.000,E1 316.053} C_DIS
LIN {X 0.075,Y -514.537,Z 1198.548,A 0.000,B 0.000,C 90.000,E1 314.595} C_DIS
LIN {X -0.137,Y -515.522,Z 1198.538,A 0.000,B 0.000,C 90.000,E1 312.852} C_DIS
LIN {X 0.243,Y -516.941,Z 1198.525,A 0.000,B 0.000,C 90.000,E1 310.458} C_DIS
LIN {X -0.221,Y -518.003,Z 1198.515,A 0.000,B 0.000,C 90.000,E1 308.749} C_DIS
LIN {X 0.267,Y -518.633,Z 1198.509,A 0.000,B 0.000,C 90.000,E1 307.523} C_DIS
LIN {X -0.129,Y -519.520,Z 1198.497,A 0.000,B 0.000,C 90.000,E1 305.518} C_DIS
LIN {X 0.050,Y -520.558,Z 1198.486,A 0.000,B 0.000,C 90.000,E1 303.452} C_DIS
LIN {X -0.018,Y -521.096,Z 1198.479,A 0.000,B 0.000,C 90.000,E1 302.291} C_DIS
LIN {X 0.304,Y -521.630,Z 1198.471,A 0.000,B 0.000,C 90.000,E1 300.797} C_DIS
LIN {X 0.037,Y -521.858,Z 1198.466,A 0.000,B 0.000,C 90.000,E1 299.951} C_DIS
LIN {X 0.097,Y -522.109,Z 1198.458,A 0.000,B 0.000,C 90.000,E1 298.487} C_DIS
LIN {X 0.043,Y -522.323,Z 1198.449,A 0.000,B 0.000,C 90.000,E1 296.744} C_DIS
LIN {X -0.070,Y -522.457,Z 1198.442,A 0.000,B 0.000,C 90.000,E1 295.591} C_DIS
LIN {X 0.120,Y -522.403,Z 1198.432,A 0.000,B 0.000,C 90.000,E1 293.823} C_DIS
LIN {X 0.250,Y -522.429,Z 1198.421,A 0.000,B 0.000,C 90.000,E1 291.770} C_DIS
LIN {X -0.133,Y -522.359,Z 1198.413,A 0.000,B 0.000,C 90.000,E1 290.355} C_DIS
LIN {X -0.053,Y -521.988,Z 1198.403,A 0.000,B 0.000,C 90.000,E1 288.598} C_DIS
LIN {X 0.083,Y -521.742,Z 1198.400,A 0.000,B 0.000,C 90.000,E1 288.000} C_DIS
LIN {X 0.119,Y -520.490,Z 1198.387,A 0.000,B 0.000,C 90.000,E1 285.662} C_DIS
LIN {X -0.275,Y -519.447,Z 1198.379,A 0.000,B 0.000,C 90.000,E1 284.245} C_DIS
LIN {X -0.184,Y -518.222,Z 1198.369,A 0.000,B 0.000,C 90.000,E1 282.479} C_DIS
LIN {X -0.144,Y -516.975,Z 1198.358,A 0.000,B 0.000,C 90.000,E1 280.423} C_DIS
LIN {X 0.093,Y -515.851,Z 1198.346,A 0.000,B 0.000,C 90.000,E1 278.341} C_DIS
LIN {X 0.279,Y -514.494,Z 1198.333,A 0.000,B 0.000,C 90.000,E1 275.967} C_DIS
LIN {X -0.176,Y -513.313,Z 1198.322,A 0.000,B 0.000,C 90.000,E1 273.955} C_DIS
LIN {X 0.162,Y -511.913,Z 1198.307,A 0.000,B 0.000,C 90.000,E1 271.260} C_DIS
LIN {X 0.094,Y -510.926,Z 1198.296,A 0.000,B 0.000,C 90.000,E1 269.198} C_DIS
LIN {X 0.097,Y -509.774,Z 1198.286,A 0.000,B 0.000,C 90.000,E1 267.421} C_DIS
LIN {X 0.163,Y -508.834,Z 1198.278,A 0.000,B 0.000,C 90.000,E1 265.931} C_DIS
LIN {X -0.162,Y -507.889,Z 1198.271,A 0.000,B 0.000,C 90.000,E1 264.780} C_DIS
LIN {X 0.008,Y -506.739,Z 1198.264,A 0.000,B 0.000,C 90.000,E1 263.571} C_DIS
LIN {X 0.163,Y -505.396,Z 1198.256,A 0.000,B 0.000,C 90.000,E1 262.064} C_DIS
LIN {X 0.100,Y -503.658,Z 1198.245,A 0.000,B 0.000,C 90.000,E1 259.982} C_DIS
LIN {X 0.086,Y -501.778,Z 1198.231,A 0.000,B 0.000,C 90.000,E1 257.589} C_DIS
LIN {X -0.078,Y -500.725,Z 1198.224,A 0.000,B 0.000,C 90.000,E1 256.408} C_DIS
LIN {X 0.280,Y -499.560,Z 1198.216,A 0.000,B 0.000,C 90.000,E1 254.866} C_DIS
LIN {X 0.114,Y -497.437,Z 1198.199,A 0.000,B 0.000,C 90.000,E1 251.873} C_DIS
LIN {X 0.123,Y -496.742,Z 1198.194,A 0.000,B 0.000,C 90.000,E1 250.967} C_DIS
LIN {X 0.231,Y -495.590,Z 1198.186,A 0.000,B 0.000,C 90.000,E1 249.444} C_DIS
LIN {X -0.103,Y -493.923,Z 1198.176,A 0.000,B 0.000,C 90.000,E1 247.667} C_DIS
LIN {X 0.075,Y -492.801,Z 1198.169,A 0.000,B 0.000,C 90.000,E1 246.433} C_DIS
LIN {X 0.256,Y -490.946,Z 1198.159,A 0.000,B 0.000,C 90.000,E1 244.588} C_DIS
LIN {X -0.103,Y -489.945,Z 1198.154,A 0.000,B 0.000,C 90.000,E1 243.717} C_DIS
LIN {X -0.201,Y -487.808,Z 1198.144,A 0.000,B 0.000,C 90.000,E1 241.897} C_DIS
LIN {X 0.084,Y -485.949,Z 1198.135,A 0.000,B 0.000,C 90.000,E1 240.333} C_DIS
LIN {X -0.284,Y -483.617,Z 1198.125,A 0.000,B 0.000,C 90.000,E1 238.535} C_DIS
LIN {X 0.024,Y -480.882,Z 1198.113,A 0.000,B 0.000,C 90.000,E1 236.342} C_DIS
LIN {X 0.057,Y -478.585,Z 1198.103,A 0.000,B 0.000,C 90.000,E1 234.482} C_DIS
LIN {X -0.063,Y -477.129,Z 1198.096,A 0.000,B 0.000,C 90.000,E1 233.256} C_DIS
LIN {X 0.092,Y -473.752,Z 1198.080,A 0.000,B 0.000,C 90.000,E1 230.436} C_DIS
LIN {X -0.166,Y -472.330,Z 1198.073,A 0.000,B 0.000,C 90.000,E1 229.218} C_DIS
LIN {X -0.082,Y -469.274,Z 1198.059,A 0.000,B 0.000,C 90.000,E1 226.701} C_DIS
LIN {X -0.203,Y -466.963,Z 1198.047,A 0.000,B 0.000,C 90.000,E1 224.514} C_DIS
LIN {X 0.010,Y -464.773,Z 1198.033,A 0.000,B 0.000,C 90.000,E1 221.962} C_DIS
LIN {X 0.083,Y -463.991,Z 1198.001,A 0.000,B 0.000,C 90.000,E1 216.251} C_DIS
LIN {X 0.169,Y -464.429,Z 1197.987,A 0.000,B 0.000,C 90.000,E1 213.706} C_DIS
LIN {X -0.065,Y -466.982,Z 1197.968,A 0.000,B 0.000,C 90.000,E1 210.256} C_DIS
LIN {X 0.079,Y -469.615,Z 1197.954,A 0.000,B 0.000,C 90.000,E1 207.719} C_DIS
LIN {X 0.023,Y -471.399,Z 1197.945,A 0.000,B 0.000,C 90.000,E1 206.155} C_DIS
LIN {X 0.115,Y -478.083,Z 1197.919,A 0.000,B 0.000,C 90.000,E1 201.461} C_DIS
LIN {X 0.020,Y -485.840,Z 1197.899,A 0.000,B 0.000,C 90.000,E1 197.764} C_DIS
LIN {X 0.147,Y -491.306,Z 1197.887,A 0.000,B 0.000,C 90.000,E1 195.607} C_DIS
LIN {X 0.162,Y -497.315,Z 1197.875,A 0.000,B 0.000,C 90.000,E1 193.480} C_DIS
LIN {X -0.267,Y -503.690,Z 1197.863,A 0.000,B 0.000,C 90.000,E1 191.422} C_DIS
LIN {X -0.192,Y -511.289,Z 1197.850,A 0.000,B 0.000,C 90.000,E1 189.029} C_DIS
LIN {X 0.003,Y -516.250,Z 1197.842,A 0.000,B 0.000,C 90.000,E1 187.530} C_DIS
LIN {X -0.214,Y -521.057,Z 1197.834,A 0.000,B 0.000,C 90.000,E1 186.087} C_DIS
LIN {X 0.125,Y -526.702,Z 1197.824,A 0.000,B 0.000,C 90.000,E1 184.302} C_DIS
LIN {X 0.040,Y -531.404,Z 1197.816,A 0.000,B 0.000,C 90.000,E1 182.865} C_DIS
LIN {X 0.010,Y -537.972,Z 1197.805,A 0.000,B 0.000,C 90.000,E1 180.859} C_DIS
LIN {X 0.141,Y -544.527,Z 1197.794,A 0.000,B 0.000,C 90.000,E1 178.854} C_DIS
LIN {X -0.105,Y -550.904,Z 1197.783,A 0.000,B 0.000,C 90.000,E1 176.906} C_DIS
LIN {X 0.089,Y -553.565,Z 1197.778,A 0.000,B 0.000,C 90.000,E1 176.045} C_DIS
LIN {X 0.061,Y -558.805,Z 1197.769,A 0.000,B 0.000,C 90.000,E1 174.375} C_DIS
LIN {X 0.000,Y -563.069,Z 1197.761,A 0.000,B 0.000,C 90.000,E1 172.996} C_DIS
LIN {X -0.012,Y -566.481,Z 1197.755,A 0.000,B 0.000,C 90.000,E1 171.894} C_DIS
LIN {X -0.261,Y -571.489,Z 1197.746,A 0.000,B 0.000,C 90.000,E1 170.274} C_DIS
LIN {X 0.153,Y -575.608,Z 1197.738,A 0.000,B 0.000,C 90.000,E1 168.870} C_DIS
LIN {X 0.309,Y -580.583,Z 1197.729,A 0.000,B 0.000,C 90.000,E1 167.229} C_DIS
LIN {X -0.242,Y -584.751,Z 1197.722,A 0.000,B 0.000,C 90.000,E1 165.936} C_DIS
LIN {X -0.017,Y -588.949,Z 1197.714,A 0.000,B 0.000,C 90.000,E1 164.574} C_DIS
LIN {X 0.274,Y -595.609,Z 1197.703,A 0.000,B 0.000,C 90.000,E1 162.417} C_DIS
LIN {X 0.289,Y -599.888,Z 1197.695,A 0.000,B 0.000,C 90.000,E1 161.094} C_DIS
LIN {X 0.212,Y -605.749,Z 1197.685,A 0.000,B 0.000,C 90.000,E1 159.263} C_DIS
LIN {X -0.022,Y -610.823,Z 1197.676,A 0.000,B 0.000,C 90.000,E1 157.720} C_DIS
LIN {X -0.132,Y -614.986,Z 1197.669,A 0.000,B 0.000,C 90.000,E1 156.433} C_DIS
LIN {X 0.306,Y -619.869,Z 1197.660,A 0.000,B 0.000,C 90.000,E1 154.845} C_DIS
LIN {X 0.015,Y -623.000,Z 1197.655,A 0.000,B 0.000,C 90.000,E1 153.845} C_DIS
LIN {X 0.055,Y -627.459,Z 1197.646,A 0.000,B 0.000,C 90.000,E1 152.308} C_DIS
LIN {X -0.101,Y -631.094,Z 1197.639,A 0.000,B 0.000,C 90.000,E1 151.051} C_DIS
LIN {X -0.151,Y -635.277,Z 1197.631,A 0.000,B 0.000,C 90.000,E1 149.537} C_DIS
LIN {X 0.161,Y -638.582,Z 1197.624,A 0.000,B 0.000,C 90.000,E1 148.250} C_DIS
LIN {X -0.351,Y -641.646,Z 1197.617,A 0.000,B 0.000,C 90.000,E1 147.041} C_DIS
LIN {X 0.062,Y -644.524,Z 1197.610,A 0.000,B 0.000,C 90.000,E1 145.754} C_DIS
LIN {X -0.070,Y -646.741,Z 1197.604,A 0.000,B 0.000,C 90.000,E1 144.769} C_DIS
LIN {X 0.175,Y -649.715,Z 1197.596,A 0.000,B 0.000,C 90.000,E1 143.256} C_DIS
LIN {X 0.085,Y -652.553,Z 1197.588,A 0.000,B 0.000,C 90.000,E1 141.778} C_DIS
LIN {X 0.342,Y -655.451,Z 1197.579,A 0.000,B 0.000,C 90.000,E1 140.275} C_DIS
LIN {X 0.145,Y -660.089,Z 1197.567,A 0.000,B 0.000,C 90.000,E1 138.081} C_DIS
LIN {X 0.077,Y -662.684,Z 1197.560,A 0.000,B 0.000,C 90.000,E1 136.863} C_DIS
LIN {X 0.022,Y -665.285,Z 1197.554,A 0.000,B 0.000,C 90.000,E1 135.648} C_DIS
LIN {X 0.030,Y -669.658,Z 1197.543,A 0.000,B 0.000,C 90.000,E1 133.704} C_DIS
LIN {X 0.156,Y -673.811,Z 1197.533,A 0.000,B 0.000,C 90.000,E1 132.000} C_DIS
LIN {X -0.015,Y -679.065,Z 1197.521,A 0.000,B 0.000,C 90.000,E1 129.850} C_DIS
LIN {X 0.355,Y -682.593,Z 1197.513,A 0.000,B 0.000,C 90.000,E1 128.382} C_DIS
LIN {X 0.004,Y -686.763,Z 1197.504,A 0.000,B 0.000,C 90.000,E1 126.744} C_DIS
LIN {X -0.116,Y -689.148,Z 1197.499,A 0.000,B 0.000,C 90.000,E1 125.804} C_DIS
LIN {X 0.349,Y -691.354,Z 1197.494,A 0.000,B 0.000,C 90.000,E1 124.818} C_DIS
LIN {X 0.130,Y -694.603,Z 1197.486,A 0.000,B 0.000,C 90.000,E1 123.420} C_DIS
LIN {X -0.100,Y -696.698,Z 1197.481,A 0.000,B 0.000,C 90.000,E1 122.498} C_DIS
LIN {X -0.007,Y -699.591,Z 1197.473,A 0.000,B 0.000,C 90.000,E1 121.082} C_DIS
LIN {X -0.140,Y -701.830,Z 1197.466,A 0.000,B 0.000,C 90.000,E1 119.922} C_DIS
LIN {X 0.290,Y -704.188,Z 1197.458,A 0.000,B 0.000,C 90.000,E1 118.487} C_DIS
LIN {X -0.140,Y -705.483,Z 1197.453,A 0.000,B 0.000,C 90.000,E1 117.590} C_DIS
LIN {X 0.107,Y -706.174,Z 1197.449,A 0.000,B 0.000,C 90.000,E1 116.873} C_DIS
LIN {X -0.299,Y -706.679,Z 1197.444,A 0.000,B 0.000,C 90.000,E1 115.976} C_DIS
LIN {X -0.004,Y -706.788,Z 1197.443,A 0.000,B 0.000,C 90.000,E1 115.720} C_DIS
LIN {X -0.062,Y -706.700,Z 1197.439,A 0.000,B 0.000,C 90.000,E1 115.027} C_DIS
LIN {X -0.118,Y -706.502,Z 1197.437,A 0.000,B 0.000,C 90.000,E1 114.567} C_DIS
LIN {X 0.174,Y -705.593,Z 1197.434,A 0.000,B 0.000,C 90.000,E1 114.079} C_DIS
LIN {X -0.182,Y -705.013,Z 1197.433,A 0.000,B 0.000,C 90.000,E1 113.875} C_DIS
LIN {X 0.244,Y -702.212,Z 1197.429,A 0.000,B 0.000,C 90.000,E1 113.259} C_DIS
LIN {X 0.107,Y -701.298,Z 1197.429,A 0.000,B 0.000,C 90.000,E1 113.153} C_DIS
LIN {X -0.080,Y -696.015,Z 1197.426,A 0.000,B 0.000,C 90.000,E1 112.717} C_DIS
LIN {X 0.162,Y -694.418,Z 1197.426,A 0.000,B 0.000,C 90.000,E1 112.589} C_DIS
LIN {X -0.238,Y -691.616,Z 1197.425,A 0.000,B 0.000,C 90.000,E1 112.514} C_DIS
LIN {X -0.227,Y -685.425,Z 1197.424,A 0.000,B 0.000,C 90.000,E1 112.333} C_DIS
LIN {X 0.168,Y -683.242,Z 1197.424,A 0.000,B 0.000,C 90.000,E1 112.280} C_DIS
LIN {X -0.045,Y -677.337,Z 1197.424,A 0.000,B 0.000,C 90.000,E1 112.280} C_DIS
LIN {X -0.083,Y -607.936,Z 1197.424,A 0.000,B 0.000,C 90.000,E1 112.280} C_DIS
LIN {X -0.056,Y -602.229,Z 1197.422,A 0.000,B 0.000,C 90.000,E1 111.897} C_DIS
LIN {X -0.285,Y -592.074,Z 1197.417,A 0.000,B 0.000,C 90.000,E1 111.099} C_DIS
LIN {X -0.307,Y -583.489,Z 1197.413,A 0.000,B 0.000,C 90.000,E1 110.429} C_DIS
LIN {X 0.078,Y -576.204,Z 1197.410,A 0.000,B 0.000,C 90.000,E1 109.812} C_DIS
LIN {X -0.138,Y -574.727,Z 1197.409,A 0.000,B 0.000,C 90.000,E1 109.631} C_DIS
LIN {X -0.181,Y -574.722,Z 1197.409,A 0.000,B 0.000,C 90.000,E1 109.631} C_DIS
LIN {X -0.138,Y -574.792,Z 1197.408,A 0.000,B 0.000,C 90.000,E1 109.504} C_DIS
LIN {X -0.122,Y -575.587,Z 1197.406,A 0.000,B 0.000,C 90.000,E1 109.141} C_DIS
LIN {X 0.095,Y -579.760,Z 1197.399,A 0.000,B 0.000,C 90.000,E1 107.764} C_DIS
LIN {X -0.212,Y -581.349,Z 1197.394,A 0.000,B 0.000,C 90.000,E1 106.985} C_DIS
LIN {X -0.167,Y -582.267,Z 1197.391,A 0.000,B 0.000,C 90.000,E1 106.441} C_DIS
LIN {X 0.106,Y -583.072,Z 1197.387,A 0.000,B 0.000,C 90.000,E1 105.607} C_DIS
LIN {X 0.157,Y -583.415,Z 1197.384,A 0.000,B 0.000,C 90.000,E1 105.064} C_DIS
LIN {X 0.058,Y -583.288,Z 1197.381,A 0.000,B 0.000,C 90.000,E1 104.537} C_DIS
LIN {X -0.038,Y -582.885,Z 1197.378,A 0.000,B 0.000,C 90.000,E1 104.008} C_DIS
LIN {X 0.198,Y -582.593,Z 1197.376,A 0.000,B 0.000,C 90.000,E1 103.716} C_DIS
LIN {X 0.234,Y -581.640,Z 1197.373,A 0.000,B 0.000,C 90.000,E1 103.175} C_DIS
LIN {X 0.129,Y -580.194,Z 1197.370,A 0.000,B 0.000,C 90.000,E1 102.647} C_DIS
LIN {X 0.014,Y -578.336,Z 1197.367,A 0.000,B 0.000,C 90.000,E1 102.119} C_DIS
LIN {X 0.003,Y -576.567,Z 1197.365,A 0.000,B 0.000,C 90.000,E1 101.715} C_DIS
LIN {X 0.218,Y -575.223,Z 1197.364,A 0.000,B 0.000,C 90.000,E1 101.422} C_DIS
LIN {X 0.303,Y -572.625,Z 1197.361,A 0.000,B 0.000,C 90.000,E1 101.007} C_DIS
LIN {X -0.168,Y -570.332,Z 1197.360,A 0.000,B 0.000,C 90.000,E1 100.782} C_DIS
LIN {X 0.262,Y -569.130,Z 1197.359,A 0.000,B 0.000,C 90.000,E1 100.602} C_DIS
LIN {X -0.173,Y -564.129,Z 1197.355,A 0.000,B 0.000,C 90.000,E1 99.962} C_DIS
LIN {X 0.031,Y -561.645,Z 1197.353,A 0.000,B 0.000,C 90.000,E1 99.557} C_DIS
LIN {X -0.119,Y -561.008,Z 1197.352,A 0.000,B 0.000,C 90.000,E1 99.434} C_DIS
LIN {X 0.138,Y -560.617,Z 1197.352,A 0.000,B 0.000,C 90.000,E1 99.265} C_DIS
LIN {X 0.042,Y -560.085,Z 1197.349,A 0.000,B 0.000,C 90.000,E1 98.859} C_DIS
LIN {X -0.094,Y -560.116,Z 1197.348,A 0.000,B 0.000,C 90.000,E1 98.568} C_DIS
LIN {X 0.050,Y -559.989,Z 1197.346,A 0.000,B 0.000,C 90.000,E1 98.276} C_DIS
LIN {X -0.263,Y -561.791,Z 1197.329,A 0.000,B 0.000,C 90.000,E1 95.277} C_DIS
LIN {X 0.283,Y -562.750,Z 1197.322,A 0.000,B 0.000,C 90.000,E1 93.841} C_DIS
LIN {X -0.104,Y -564.067,Z 1197.311,A 0.000,B 0.000,C 90.000,E1 91.949} C_DIS
LIN {X -0.112,Y -565.096,Z 1197.303,A 0.000,B 0.000,C 90.000,E1 90.573} C_DIS
LIN {X 0.114,Y -566.497,Z 1197.292,A 0.000,B 0.000,C 90.000,E1 88.625} C_DIS
LIN {X -0.156,Y -567.903,Z 1197.282,A 0.000,B 0.000,C 90.000,E1 86.731} C_DIS
LIN {X 0.063,Y -569.159,Z 1197.273,A 0.000,B 0.000,C 90.000,E1 85.065} C_DIS
LIN {X 0.181,Y -570.132,Z 1197.265,A 0.000,B 0.000,C 90.000,E1 83.685} C_DIS
LIN {X -0.004,Y -571.348,Z 1197.256,A 0.000,B 0.000,C 90.000,E1 82.064} C_DIS
LIN {X 0.018,Y -572.079,Z 1197.250,A 0.000,B 0.000,C 90.000,E1 80.971} C_DIS
LIN {X -0.043,Y -573.118,Z 1197.241,A 0.000,B 0.000,C 90.000,E1 79.342} C_DIS
LIN {X -0.171,Y -573.942,Z 1197.233,A 0.000,B 0.000,C 90.000,E1 77.993} C_DIS
LIN {X -0.081,Y -574.763,Z 1197.224,A 0.000,B 0.000,C 90.000,E1 76.353} C_DIS
LIN {X -0.048,Y -575.770,Z 1197.214,A 0.000,B 0.000,C 90.000,E1 74.448} C_DIS
LIN {X 0.013,Y -576.734,Z 1197.203,A 0.000,B 0.000,C 90.000,E1 72.543} C_DIS
LIN {X 0.064,Y -577.701,Z 1197.194,A 0.000,B 0.000,C 90.000,E1 70.913} C_DIS
LIN {X -0.030,Y -579.007,Z 1197.183,A 0.000,B 0.000,C 90.000,E1 69.028} C_DIS
LIN {X -0.043,Y -580.784,Z 1197.172,A 0.000,B 0.000,C 90.000,E1 66.869} C_DIS
LIN {X -0.066,Y -581.892,Z 1197.166,A 0.000,B 0.000,C 90.000,E1 65.793} C_DIS
LIN {X 0.071,Y -583.614,Z 1197.155,A 0.000,B 0.000,C 90.000,E1 63.896} C_DIS
LIN {X 0.109,Y -585.254,Z 1197.146,A 0.000,B 0.000,C 90.000,E1 62.281} C_DIS
LIN {X 0.176,Y -586.854,Z 1197.137,A 0.000,B 0.000,C 90.000,E1 60.667} C_DIS
LIN {X -0.014,Y -587.849,Z 1197.131,A 0.000,B 0.000,C 90.000,E1 59.616} C_DIS
LIN {X -0.012,Y -588.979,Z 1197.124,A 0.000,B 0.000,C 90.000,E1 58.280} C_DIS
LIN {X -0.295,Y -590.283,Z 1197.115,A 0.000,B 0.000,C 90.000,E1 56.707} C_DIS
LIN {X -0.218,Y -591.440,Z 1197.106,A 0.000,B 0.000,C 90.000,E1 55.102} C_DIS
LIN {X -0.117,Y -592.663,Z 1197.097,A 0.000,B 0.000,C 90.000,E1 53.497} C_DIS
LIN {X -0.120,Y -593.781,Z 1197.088,A 0.000,B 0.000,C 90.000,E1 51.904} C_DIS
LIN {X 0.054,Y -594.555,Z 1197.081,A 0.000,B 0.000,C 90.000,E1 50.561} C_DIS
LIN {X 0.245,Y -595.301,Z 1197.074,A 0.000,B 0.000,C 90.000,E1 49.218} C_DIS
LIN {X -0.005,Y -595.752,Z 1197.066,A 0.000,B 0.000,C 90.000,E1 47.919} C_DIS
LIN {X -0.030,Y -596.010,Z 1197.060,A 0.000,B 0.000,C 90.000,E1 46.863} C_DIS
LIN {X -0.083,Y -596.132,Z 1197.055,A 0.000,B 0.000,C 90.000,E1 45.810} C_DIS
LIN {X -0.127,Y -596.088,Z 1197.049,A 0.000,B 0.000,C 90.000,E1 44.757} C_DIS
LIN {X 0.035,Y -595.738,Z 1197.041,A 0.000,B 0.000,C 90.000,E1 43.419} C_DIS
LIN {X 0.205,Y -595.364,Z 1197.037,A 0.000,B 0.000,C 90.000,E1 42.609} C_DIS
LIN {X -0.037,Y -594.908,Z 1197.032,A 0.000,B 0.000,C 90.000,E1 41.838} C_DIS
LIN {X -0.301,Y -593.965,Z 1197.025,A 0.000,B 0.000,C 90.000,E1 40.539} C_DIS
LIN {X -0.107,Y -593.355,Z 1197.021,A 0.000,B 0.000,C 90.000,E1 39.725} C_DIS
LIN {X -0.163,Y -592.366,Z 1197.015,A 0.000,B 0.000,C 90.000,E1 38.669} C_DIS
LIN {X 0.073,Y -590.778,Z 1197.007,A 0.000,B 0.000,C 90.000,E1 37.317} C_DIS
LIN {X 0.227,Y -589.671,Z 1197.003,A 0.000,B 0.000,C 90.000,E1 36.503} C_DIS
LIN {X 0.015,Y -588.481,Z 1196.999,A 0.000,B 0.000,C 90.000,E1 35.724} C_DIS
LIN {X -0.158,Y -585.934,Z 1196.991,A 0.000,B 0.000,C 90.000,E1 34.405} C_DIS
LIN {X 0.075,Y -583.934,Z 1196.987,A 0.000,B 0.000,C 90.000,E1 33.579} C_DIS
LIN {X 0.285,Y -581.692,Z 1196.982,A 0.000,B 0.000,C 90.000,E1 32.752} C_DIS
LIN {X -0.331,Y -579.144,Z 1196.978,A 0.000,B 0.000,C 90.000,E1 32.005} C_DIS
LIN {X -0.174,Y -578.220,Z 1196.976,A 0.000,B 0.000,C 90.000,E1 31.720} C_DIS
LIN {X 0.296,Y -573.998,Z 1196.970,A 0.000,B 0.000,C 90.000,E1 30.590} C_DIS
LIN {X 0.094,Y -570.267,Z 1196.966,A 0.000,B 0.000,C 90.000,E1 29.795} C_DIS
LIN {X -0.251,Y -567.536,Z 1196.963,A 0.000,B 0.000,C 90.000,E1 29.283} C_DIS
LIN {X 0.146,Y -562.382,Z 1196.957,A 0.000,B 0.000,C 90.000,E1 28.281} C_DIS
LIN {X 0.046,Y -557.451,Z 1196.953,A 0.000,B 0.000,C 90.000,E1 27.462} C_DIS
LIN {X 0.155,Y -552.141,Z 1196.948,A 0.000,B 0.000,C 90.000,E1 26.616} C_DIS
LIN {X 0.079,Y -547.297,Z 1196.944,A 0.000,B 0.000,C 90.000,E1 25.924} C_DIS
LIN {X 0.321,Y -543.060,Z 1196.941,A 0.000,B 0.000,C 90.000,E1 25.335} C_DIS
LIN {X -0.186,Y -538.533,Z 1196.938,A 0.000,B 0.000,C 90.000,E1 24.823} C_DIS
LIN {X -0.035,Y -531.397,Z 1196.933,A 0.000,B 0.000,C 90.000,E1 23.951} C_DIS
LIN {X 0.228,Y -525.038,Z 1196.929,A 0.000,B 0.000,C 90.000,E1 23.206} C_DIS
LIN {X -0.042,Y -517.047,Z 1196.924,A 0.000,B 0.000,C 90.000,E1 22.386} C_DIS
LIN {X 0.012,Y -507.534,Z 1196.919,A 0.000,B 0.000,C 90.000,E1 21.408} C_DIS
LIN {X -0.034,Y -499.236,Z 1196.915,A 0.000,B 0.000,C 90.000,E1 20.610} C_DIS
LIN {X 0.076,Y -493.635,Z 1196.912,A 0.000,B 0.000,C 90.000,E1 20.066} C_DIS
LIN {X 0.054,Y -483.503,Z 1196.906,A 0.000,B 0.000,C 90.000,E1 19.141} C_DIS
LIN {X 0.025,Y -476.195,Z 1196.903,A 0.000,B 0.000,C 90.000,E1 18.489} C_DIS
LIN {X -0.239,Y -466.203,Z 1196.898,A 0.000,B 0.000,C 90.000,E1 17.638} C_DIS
LIN {X -0.154,Y -447.214,Z 1196.888,A 0.000,B 0.000,C 90.000,E1 15.898} C_DIS
LIN {X -0.107,Y -426.911,Z 1196.877,A 0.000,B 0.000,C 90.000,E1 13.883} C_DIS
LIN {X 0.032,Y -413.326,Z 1196.869,A 0.000,B 0.000,C 90.000,E1 12.355} C_DIS
LIN {X 0.128,Y -402.407,Z 1196.861,A 0.000,B 0.000,C 90.000,E1 11.007} C_DIS
LIN {X 0.126,Y -399.768,Z 1196.859,A 0.000,B 0.000,C 90.000,E1 10.658} C_DIS
LIN {X 0.210,Y -395.604,Z 1196.856,A 0.000,B 0.000,C 90.000,E1 10.018} C_DIS
LIN {X -0.188,Y -393.528,Z 1196.853,A 0.000,B 0.000,C 90.000,E1 9.613} C_DIS
LIN {X 0.118,Y -393.174,Z 1196.852,A 0.000,B 0.000,C 90.000,E1 9.265} C_DIS
LIN {X 0.080,Y -393.174,Z 1196.852,A 0.000,B 0.000,C 90.000,E1 9.265} C_DIS
LIN {X 0.057,Y -394.071,Z 1196.849,A 0.000,B 0.000,C 90.000,E1 8.803} C_DIS
LIN {X 0.012,Y -396.942,Z 1196.845,A 0.000,B 0.000,C 90.000,E1 8.106} C_DIS
LIN {X -0.057,Y -400.204,Z 1196.842,A 0.000,B 0.000,C 90.000,E1 7.587} C_DIS
LIN {X -0.042,Y -401.356,Z 1196.841,A 0.000,B 0.000,C 90.000,E1 7.409} C_DIS
LIN {X -0.075,Y -402.743,Z 1196.840,A 0.000,B 0.000,C 90.000,E1 7.239} C_DIS
LIN {X 0.039,Y -405.839,Z 1196.838,A 0.000,B 0.000,C 90.000,E1 6.891} C_DIS
LIN {X -0.046,Y -411.416,Z 1196.836,A 0.000,B 0.000,C 90.000,E1 6.429} C_DIS
LIN {X -0.145,Y -425.714,Z 1196.830,A 0.000,B 0.000,C 90.000,E1 5.334} C_DIS
LIN {X -0.091,Y -438.487,Z 1196.824,A 0.000,B 0.000,C 90.000,E1 4.359} C_DIS
LIN {X -0.217,Y -451.135,Z 1196.819,A 0.000,B 0.000,C 90.000,E1 3.440} C_DIS
LIN {X 0.109,Y -465.494,Z 1196.813,A 0.000,B 0.000,C 90.000,E1 2.350} C_DIS
LIN {X 0.010,Y -473.169,Z 1196.810,A 0.000,B 0.000,C 90.000,E1 1.776} C_DIS
LIN {X -0.231,Y -479.283,Z 1196.807,A 0.000,B 0.000,C 90.000,E1 1.318} C_DIS
LIN {X -0.094,Y -485.281,Z 1196.804,A 0.000,B 0.000,C 90.000,E1 0.802} C_DIS
LIN {X -0.128,Y -491.130,Z 1196.802,A 0.000,B 0.000,C 90.000,E1 0.286} C_DIS
LIN {X 0.013,Y -497.498,Z 1196.798,A 0.000,B 0.000,C 90.000,E1 359.656} C_DIS
LIN {X -0.069,Y -504.244,Z 1196.794,A 0.000,B 0.000,C 90.000,E1 358.969} C_DIS
LIN {X -0.203,Y -511.782,Z 1196.789,A 0.000,B 0.000,C 90.000,E1 358.108} C_DIS
LIN {X 0.145,Y -516.610,Z 1196.786,A 0.000,B 0.000,C 90.000,E1 357.478} C_DIS
LIN {X 0.269,Y -522.090,Z 1196.782,A 0.000,B 0.000,C 90.000,E1 356.731} C_DIS
LIN {X -0.116,Y -527.107,Z 1196.778,A 0.000,B 0.000,C 90.000,E1 356.045} C_DIS
LIN {X 0.103,Y -531.560,Z 1196.774,A 0.000,B 0.000,C 90.000,E1 355.298} C_DIS
LIN {X 0.106,Y -534.932,Z 1196.771,A 0.000,B 0.000,C 90.000,E1 354.723} C_DIS
LIN {X -0.137,Y -538.586,Z 1196.767,A 0.000,B 0.000,C 90.000,E1 354.033} C_DIS
LIN {X 0.249,Y -541.970,Z 1196.763,A 0.000,B 0.000,C 90.000,E1 353.280} C_DIS
LIN {X 0.054,Y -543.891,Z 1196.760,A 0.000,B 0.000,C 90.000,E1 352.875} C_DIS
LIN {X -0.295,Y -548.410,Z 1196.754,A 0.000,B 0.000,C 90.000,E1 351.781} C_DIS
LIN {X 0.010,Y -551.393,Z 1196.750,A 0.000,B 0.000,C 90.000,E1 350.905} C_DIS
LIN {X 0.265,Y -554.079,Z 1196.745,A 0.000,B 0.000,C 90.000,E1 350.038} C_DIS
LIN {X 0.232,Y -557.310,Z 1196.739,A 0.000,B 0.000,C 90.000,E1 348.926} C_DIS
LIN {X -0.010,Y -559.560,Z 1196.734,A 0.000,B 0.000,C 90.000,E1 348.117} C_DIS
LIN {X 0.001,Y -561.623,Z 1196.729,A 0.000,B 0.000,C 90.000,E1 347.285} C_DIS
LIN {X -0.082,Y -563.613,Z 1196.725,A 0.000,B 0.000,C 90.000,E1 346.464} C_DIS
LIN {X -0.064,Y -567.227,Z 1196.716,A 0.000,B 0.000,C 90.000,E1 344.810} C_DIS
LIN {X 0.218,Y -569.406,Z 1196.709,A 0.000,B 0.000,C 90.000,E1 343.685} C_DIS
LIN {X -0.225,Y -571.997,Z 1196.702,A 0.000,B 0.000,C 90.000,E1 342.362} C_DIS
LIN {X -0.258,Y -573.889,Z 1196.696,A 0.000,B 0.000,C 90.000,E1 341.275} C_DIS
LIN {X -0.266,Y -575.544,Z 1196.690,A 0.000,B 0.000,C 90.000,E1 340.188} C_DIS
LIN {X -0.057,Y -576.943,Z 1196.684,A 0.000,B 0.000,C 90.000,E1 339.082} C_DIS
LIN {X -0.206,Y -577.740,Z 1196.679,A 0.000,B 0.000,C 90.000,E1 338.284} C_DIS
LIN {X 0.034,Y -578.512,Z 1196.673,A 0.000,B 0.000,C 90.000,E1 337.177} C_DIS
LIN {X 0.122,Y -578.701,Z 1196.669,A 0.000,B 0.000,C 90.000,E1 336.357} C_DIS
LIN {X -0.167,Y -578.719,Z 1196.666,A 0.000,B 0.000,C 90.000,E1 335.845} C_DIS
LIN {X -0.068,Y -578.375,Z 1196.661,A 0.000,B 0.000,C 90.000,E1 335.025} C_DIS
LIN {X 0.169,Y -577.999,Z 1196.658,A 0.000,B 0.000,C 90.000,E1 334.460} C_DIS
LIN {X 0.256,Y -577.037,Z 1196.654,A 0.000,B 0.000,C 90.000,E1 333.640} C_DIS
LIN {X -0.188,Y -575.726,Z 1196.649,A 0.000,B 0.000,C 90.000,E1 332.871} C_DIS
LIN {X 0.132,Y -573.992,Z 1196.645,A 0.000,B 0.000,C 90.000,E1 332.025} C_DIS
LIN {X -0.068,Y -571.994,Z 1196.640,A 0.000,B 0.000,C 90.000,E1 331.229} C_DIS
LIN {X 0.102,Y -570.476,Z 1196.637,A 0.000,B 0.000,C 90.000,E1 330.667} C_DIS
LIN {X 0.041,Y -568.627,Z 1196.634,A 0.000,B 0.000,C 90.000,E1 330.127} C_DIS
LIN {X -0.028,Y -566.444,Z 1196.631,A 0.000,B 0.000,C 90.000,E1 329.587} C_DIS
LIN {X 0.376,Y -563.857,Z 1196.628,A 0.000,B 0.000,C 90.000,E1 328.997} C_DIS
LIN {X 0.270,Y -560.945,Z 1196.625,A 0.000,B 0.000,C 90.000,E1 328.456} C_DIS
LIN {X 0.037,Y -556.570,Z 1196.621,A 0.000,B 0.000,C 90.000,E1 327.788} C_DIS
LIN {X -0.233,Y -551.653,Z 1196.617,A 0.000,B 0.000,C 90.000,E1 327.120} C_DIS
LIN {X -0.119,Y -547.527,Z 1196.614,A 0.000,B 0.000,C 90.000,E1 326.548} C_DIS
LIN {X 0.284,Y -541.829,Z 1196.610,A 0.000,B 0.000,C 90.000,E1 325.801} C_DIS
LIN {X -0.046,Y -533.449,Z 1196.605,A 0.000,B 0.000,C 90.000,E1 324.848} C_DIS
LIN {X 0.133,Y -527.285,Z 1196.601,A 0.000,B 0.000,C 90.000,E1 324.116} C_DIS
LIN {X -0.119,Y -522.458,Z 1196.598,A 0.000,B 0.000,C 90.000,E1 323.577} C_DIS
LIN {X -0.019,Y -519.143,Z 1196.595,A 0.000,B 0.000,C 90.000,E1 323.130} C_DIS
LIN {X 0.033,Y -516.803,Z 1196.593,A 0.000,B 0.000,C 90.000,E1 322.763} C_DIS
LIN {X -0.151,Y -515.975,Z 1196.592,A 0.000,B 0.000,C 90.000,E1 322.637} C_DIS
LIN {X -0.028,Y -513.769,Z 1196.590,A 0.000,B 0.000,C 90.000,E1 322.145} C_DIS
LIN {X -0.010,Y -512.242,Z 1196.586,A 0.000,B 0.000,C 90.000,E1 321.537} C_DIS
LIN {X 0.030,Y -511.816,Z 1196.584,A 0.000,B 0.000,C 90.000,E1 321.090} C_DIS
LIN {X -0.136,Y -511.656,Z 1196.581,A 0.000,B 0.000,C 90.000,E1 320.517} C_DIS
LIN {X -0.053,Y -513.157,Z 1196.564,A 0.000,B 0.000,C 90.000,E1 317.553} C_DIS
LIN {X 0.167,Y -513.986,Z 1196.556,A 0.000,B 0.000,C 90.000,E1 316.053} C_DIS
LIN {X 0.035,Y -514.824,Z 1196.548,A 0.000,B 0.000,C 90.000,E1 314.595} C_DIS
LIN {X -0.087,Y -515.675,Z 1196.540,A 0.000,B 0.000,C 90.000,E1 313.137} C_DIS
LIN {X -0.048,Y -517.080,Z 1196.527,A 0.000,B 0.000,C 90.000,E1 310.782} C_DIS
LIN {X 0.023,Y -517.789,Z 1196.520,A 0.000,B 0.000,C 90.000,E1 309.600} C_DIS
LIN {X -0.037,Y -518.675,Z 1196.512,A 0.000,B 0.000,C 90.000,E1 308.141} C_DIS
LIN {X 0.144,Y -519.241,Z 1196.505,A 0.000,B 0.000,C 90.000,E1 306.950} C_DIS
LIN {X -0.185,Y -520.076,Z 1196.496,A 0.000,B 0.000,C 90.000,E1 305.231} C_DIS
LIN {X 0.004,Y -521.093,Z 1196.484,A 0.000,B 0.000,C 90.000,E1 303.166} C_DIS
LIN {X -0.003,Y -521.498,Z 1196.479,A 0.000,B 0.000,C 90.000,E1 302.291} C_DIS
LIN {X -0.123,Y -522.054,Z 1196.471,A 0.000,B 0.000,C 90.000,E1 300.846} C_DIS
LIN {X 0.064,Y -522.293,Z 1196.466,A 0.000,B 0.000,C 90.000,E1 299.951} C_DIS
LIN {X 0.131,Y -522.551,Z 1196.458,A 0.000,B 0.000,C 90.000,E1 298.487} C_DIS
LIN {X -0.059,Y -522.759,Z 1196.450,A 0.000,B 0.000,C 90.000,E1 297.052} C_DIS
LIN {X -0.018,Y -522.932,Z 1196.442,A 0.000,B 0.000,C 90.000,E1 295.591} C_DIS
LIN {X 0.026,Y -522.919,Z 1196.434,A 0.000,B 0.000,C 90.000,E1 294.131} C_DIS
LIN {X 0.166,Y -522.859,Z 1196.423,A 0.000,B 0.000,C 90.000,E1 292.078} C_DIS
LIN {X -0.051,Y -522.795,Z 1196.413,A 0.000,B 0.000,C 90.000,E1 290.355} C_DIS
LIN {X 0.040,Y -522.480,Z 1196.403,A 0.000,B 0.000,C 90.000,E1 288.598} C_DIS
LIN {X -0.168,Y -522.058,Z 1196.399,A 0.000,B 0.000,C 90.000,E1 287.747} C_DIS
LIN {X 0.093,Y -521.169,Z 1196.389,A 0.000,B 0.000,C 90.000,E1 285.969} C_DIS
LIN {X -0.148,Y -520.412,Z 1196.382,A 0.000,B 0.000,C 90.000,E1 284.828} C_DIS
LIN {X -0.048,Y -518.976,Z 1196.371,A 0.000,B 0.000,C 90.000,E1 282.771} C_DIS
LIN {X -0.093,Y -517.501,Z 1196.358,A 0.000,B 0.000,C 90.000,E1 280.433} C_DIS
LIN {X -0.260,Y -516.373,Z 1196.347,A 0.000,B 0.000,C 90.000,E1 278.398} C_DIS
LIN {X -0.003,Y -515.395,Z 1196.337,A 0.000,B 0.000,C 90.000,E1 276.606} C_DIS
LIN {X -0.175,Y -514.667,Z 1196.330,A 0.000,B 0.000,C 90.000,E1 275.448} C_DIS
LIN {X 0.013,Y -513.839,Z 1196.322,A 0.000,B 0.000,C 90.000,E1 273.955} C_DIS
LIN {X -0.144,Y -512.462,Z 1196.307,A 0.000,B 0.000,C 90.000,E1 271.318} C_DIS
LIN {X -0.197,Y -511.468,Z 1196.296,A 0.000,B 0.000,C 90.000,E1 269.255} C_DIS
LIN {X 0.062,Y -510.936,Z 1196.291,A 0.000,B 0.000,C 90.000,E1 268.339} C_DIS
LIN {X -0.007,Y -509.619,Z 1196.279,A 0.000,B 0.000,C 90.000,E1 266.274} C_DIS
LIN {X 0.191,Y -508.744,Z 1196.273,A 0.000,B 0.000,C 90.000,E1 265.065} C_DIS
LIN {X -0.127,Y -507.605,Z 1196.266,A 0.000,B 0.000,C 90.000,E1 263.913} C_DIS
LIN {X -0.139,Y -505.949,Z 1196.256,A 0.000,B 0.000,C 90.000,E1 262.129} C_DIS
LIN {X -0.115,Y -504.217,Z 1196.245,A 0.000,B 0.000,C 90.000,E1 260.038} C_DIS
LIN {X 0.082,Y -503.003,Z 1196.236,A 0.000,B 0.000,C 90.000,E1 258.522} C_DIS
LIN {X -0.240,Y -501.828,Z 1196.228,A 0.000,B 0.000,C 90.000,E1 257.061} C_DIS
LIN {X -0.018,Y -500.093,Z 1196.216,A 0.000,B 0.000,C 90.000,E1 254.936} C_DIS
LIN {X -0.142,Y -498.283,Z 1196.203,A 0.000,B 0.000,C 90.000,E1 252.543} C_DIS
LIN {X -0.068,Y -497.488,Z 1196.196,A 0.000,B 0.000,C 90.000,E1 251.329} C_DIS
LIN {X -0.061,Y -496.043,Z 1196.186,A 0.000,B 0.000,C 90.000,E1 249.518} C_DIS
LIN {X 0.252,Y -494.390,Z 1196.176,A 0.000,B 0.000,C 90.000,E1 247.667} C_DIS
LIN {X -0.017,Y -493.253,Z 1196.169,A 0.000,B 0.000,C 90.000,E1 246.485} C_DIS
LIN {X -0.030,Y -491.422,Z 1196.159,A 0.000,B 0.000,C 90.000,E1 244.665} C_DIS
LIN {X 0.098,Y -489.667,Z 1196.151,A 0.000,B 0.000,C 90.000,E1 243.127} C_DIS
LIN {X 0.180,Y -488.233,Z 1196.144,A 0.000,B 0.000,C 90.000,E1 241.897} C_DIS
LIN {X 0.051,Y -486.353,Z 1196.135,A 0.000,B 0.000,C 90.000,E1 240.383} C_DIS
LIN {X 0.110,Y -484.015,Z 1196.125,A 0.000,B 0.000,C 90.000,E1 238.535} C_DIS
LIN {X -0.051,Y -481.665,Z 1196.115,A 0.000,B 0.000,C 90.000,E1 236.707} C_DIS
LIN {X -0.202,Y -478.920,Z 1196.103,A 0.000,B 0.000,C 90.000,E1 234.562} C_DIS
LIN {X -0.135,Y -477.028,Z 1196.094,A 0.000,B 0.000,C 90.000,E1 233.004} C_DIS
LIN {X -0.155,Y -474.019,Z 1196.081,A 0.000,B 0.000,C 90.000,E1 230.517} C_DIS
LIN {X 0.036,Y -472.170,Z 1196.072,A 0.000,B 0.000,C 90.000,E1 228.933} C_DIS
LIN {X 0.005,Y -469.473,Z 1196.060,A 0.000,B 0.000,C 90.000,E1 226.743} C_DIS
LIN {X 0.299,Y -466.750,Z 1196.046,A 0.000,B 0.000,C 90.000,E1 224.190} C_DIS
LIN {X 0.130,Y -464.814,Z 1196.033,A 0.000,B 0.000,C 90.000,E1 222.000} C_DIS
LIN {X 0.069,Y -463.688,Z 1196.011,A 0.000,B 0.000,C 90.000,E1 217.890} C_DIS
LIN {X -0.110,Y -463.882,Z 1196.000,A 0.000,B 0.000,C 90.000,E1 216.011} C_DIS
LIN {X -0.052,Y -464.215,Z 1195.988,A 0.000,B 0.000,C 90.000,E1 213.785} C_DIS
LIN {X 0.204,Y -466.430,Z 1195.970,A 0.000,B 0.000,C 90.000,E1 210.590} C_DIS
LIN {X 0.011,Y -469.610,Z 1195.953,A 0.000,B 0.000,C 90.000,E1 207.462} C_DIS
LIN {X -0.045,Y -471.394,Z 1195.944,A 0.000,B 0.000,C 90.000,E1 205.899} C_DIS
LIN {X -0.115,Y -477.713,Z 1195.920,A 0.000,B 0.000,C 90.000,E1 201.535} C_DIS
LIN {X -0.064,Y -485.468,Z 1195.899,A 0.000,B 0.000,C 90.000,E1 197.819} C_DIS
LIN {X 0.047,Y -490.990,Z 1195.887,A 0.000,B 0.000,C 90.000,E1 195.662} C_DIS
LIN {X 0.048,Y -497.026,Z 1195.875,A 0.000,B 0.000,C 90.000,E1 193.536} C_DIS
LIN {X 0.100,Y -503.437,Z 1195.864,A 0.000,B 0.000,C 90.000,E1 191.422} C_DIS
LIN {X 0.173,Y -511.113,Z 1195.850,A 0.000,B 0.000,C 90.000,E1 189.029} C_DIS
LIN {X -0.144,Y -516.094,Z 1195.842,A 0.000,B 0.000,C 90.000,E1 187.587} C_DIS
LIN {X 0.140,Y -521.859,Z 1195.832,A 0.000,B 0.000,C 90.000,E1 185.796} C_DIS
LIN {X -0.070,Y -528.492,Z 1195.821,A 0.000,B 0.000,C 90.000,E1 183.784} C_DIS
LIN {X -0.156,Y -533.196,Z 1195.813,A 0.000,B 0.000,C 90.000,E1 182.350} C_DIS
LIN {X -0.148,Y -538.855,Z 1195.803,A 0.000,B 0.000,C 90.000,E1 180.630} C_DIS
LIN {X -0.027,Y -544.530,Z 1195.794,A 0.000,B 0.000,C 90.000,E1 178.912} C_DIS
LIN {X 0.227,Y -550.044,Z 1195.785,A 0.000,B 0.000,C 90.000,E1 177.192} C_DIS
LIN {X -0.080,Y -553.667,Z 1195.778,A 0.000,B 0.000,C 90.000,E1 176.102} C_DIS
LIN {X -0.229,Y -558.095,Z 1195.771,A 0.000,B 0.000,C 90.000,E1 174.723} C_DIS
LIN {X -0.241,Y -562.458,Z 1195.763,A 0.000,B 0.000,C 90.000,E1 173.337} C_DIS
LIN {X -0.171,Y -566.749,Z 1195.755,A 0.000,B 0.000,C 90.000,E1 171.951} C_DIS
LIN {X -0.124,Y -570.149,Z 1195.749,A 0.000,B 0.000,C 90.000,E1 170.849} C_DIS
LIN {X -0.197,Y -575.197,Z 1195.740,A 0.000,B 0.000,C 90.000,E1 169.218} C_DIS
LIN {X 0.048,Y -581.072,Z 1195.729,A 0.000,B 0.000,C 90.000,E1 167.297} C_DIS
LIN {X 0.203,Y -585.240,Z 1195.722,A 0.000,B 0.000,C 90.000,E1 165.936} C_DIS
LIN {X -0.128,Y -589.464,Z 1195.715,A 0.000,B 0.000,C 90.000,E1 164.629} C_DIS
LIN {X -0.262,Y -595.352,Z 1195.704,A 0.000,B 0.000,C 90.000,E1 162.779} C_DIS
LIN {X 0.212,Y -600.453,Z 1195.695,A 0.000,B 0.000,C 90.000,E1 161.148} C_DIS
LIN {X -0.060,Y -606.269,Z 1195.685,A 0.000,B 0.000,C 90.000,E1 159.337} C_DIS
LIN {X -0.295,Y -611.260,Z 1195.677,A 0.000,B 0.000,C 90.000,E1 157.794} C_DIS
LIN {X -0.162,Y -615.390,Z 1195.669,A 0.000,B 0.000,C 90.000,E1 156.485} C_DIS
LIN {X 0.040,Y -619.427,Z 1195.662,A 0.000,B 0.000,C 90.000,E1 155.177} C_DIS
LIN {X 0.010,Y -623.309,Z 1195.655,A 0.000,B 0.000,C 90.000,E1 153.896} C_DIS
LIN {X 0.063,Y -627.696,Z 1195.646,A 0.000,B 0.000,C 90.000,E1 152.359} C_DIS
LIN {X -0.412,Y -630.621,Z 1195.641,A 0.000,B 0.000,C 90.000,E1 151.385} C_DIS
LIN {X 0.072,Y -634.766,Z 1195.632,A 0.000,B 0.000,C 90.000,E1 149.822} C_DIS
LIN {X -0.004,Y -637.410,Z 1195.627,A 0.000,B 0.000,C 90.000,E1 148.820} C_DIS
LIN {X -0.202,Y -640.529,Z 1195.620,A 0.000,B 0.000,C 90.000,E1 147.582} C_DIS
LIN {X 0.150,Y -642.897,Z 1195.614,A 0.000,B 0.000,C 90.000,E1 146.548} C_DIS
LIN {X 0.056,Y -645.661,Z 1195.607,A 0.000,B 0.000,C 90.000,E1 145.308} C_DIS
LIN {X 0.048,Y -647.237,Z 1195.603,A 0.000,B 0.000,C 90.000,E1 144.562} C_DIS
LIN {X -0.136,Y -649.685,Z 1195.596,A 0.000,B 0.000,C 90.000,E1 143.336} C_DIS
LIN {X -0.273,Y -652.037,Z 1195.589,A 0.000,B 0.000,C 90.000,E1 142.110} C_DIS
LIN {X 0.022,Y -655.371,Z 1195.580,A 0.000,B 0.000,C 90.000,E1 140.356} C_DIS
LIN {X -0.184,Y -659.990,Z 1195.568,A 0.000,B 0.000,C 90.000,E1 138.162} C_DIS
LIN {X 0.199,Y -662.580,Z 1195.561,A 0.000,B 0.000,C 90.000,E1 136.905} C_DIS
LIN {X -0.306,Y -664.670,Z 1195.555,A 0.000,B 0.000,C 90.000,E1 135.972} C_DIS
LIN {X -0.309,Y -669.531,Z 1195.543,A 0.000,B 0.000,C 90.000,E1 133.785} C_DIS
LIN {X -0.170,Y -674.232,Z 1195.532,A 0.000,B 0.000,C 90.000,E1 131.838} C_DIS
LIN {X 0.157,Y -678.901,Z 1195.522,A 0.000,B 0.000,C 90.000,E1 129.886} C_DIS
LIN {X 0.004,Y -682.441,Z 1195.514,A 0.000,B 0.000,C 90.000,E1 128.463} C_DIS
LIN {X 0.061,Y -686.608,Z 1195.505,A 0.000,B 0.000,C 90.000,E1 126.790} C_DIS
LIN {X -0.068,Y -688.992,Z 1195.499,A 0.000,B 0.000,C 90.000,E1 125.851} C_DIS
LIN {X 0.356,Y -690.683,Z 1195.495,A 0.000,B 0.000,C 90.000,E1 125.105} C_DIS
LIN {X -0.224,Y -694.477,Z 1195.486,A 0.000,B 0.000,C 90.000,E1 123.499} C_DIS
LIN {X -0.080,Y -696.577,Z 1195.481,A 0.000,B 0.000,C 90.000,E1 122.546} C_DIS
LIN {X 0.002,Y -699.481,Z 1195.473,A 0.000,B 0.000,C 90.000,E1 121.131} C_DIS
LIN {X 0.119,Y -701.720,Z 1195.467,A 0.000,B 0.000,C 90.000,E1 119.951} C_DIS
LIN {X -0.056,Y -704.068,Z 1195.459,A 0.000,B 0.000,C 90.000,E1 118.565} C_DIS
LIN {X -0.156,Y -705.388,Z 1195.453,A 0.000,B 0.000,C 90.000,E1 117.641} C_DIS
LIN {X 0.085,Y -706.099,Z 1195.450,A 0.000,B 0.000,C 90.000,E1 116.924} C_DIS
LIN {X 0.309,Y -706.630,Z 1195.444,A 0.000,B 0.000,C 90.000,E1 115.976} C_DIS
LIN {X -0.046,Y -706.755,Z 1195.442,A 0.000,B 0.000,C 90.000,E1 115.540} C_DIS
LIN {X -0.094,Y -706.717,Z 1195.439,A 0.000,B 0.000,C 90.000,E1 115.079} C_DIS
LIN {X 0.196,Y -706.506,Z 1195.437,A 0.000,B 0.000,C 90.000,E1 114.591} C_DIS
LIN {X -0.153,Y -706.167,Z 1195.435,A 0.000,B 0.000,C 90.000,E1 114.387} C_DIS
LIN {X 0.140,Y -705.189,Z 1195.433,A 0.000,B 0.000,C 90.000,E1 113.898} C_DIS
LIN {X -0.073,Y -702.488,Z 1195.430,A 0.000,B 0.000,C 90.000,E1 113.334} C_DIS
LIN {X 0.067,Y -701.716,Z 1195.429,A 0.000,B 0.000,C 90.000,E1 113.206} C_DIS
LIN {X 0.204,Y -700.569,Z 1195.428,A 0.000,B 0.000,C 90.000,E1 113.078} C_DIS
LIN {X 0.107,Y -695.247,Z 1195.426,A 0.000,B 0.000,C 90.000,E1 112.642} C_DIS
LIN {X 0.353,Y -693.176,Z 1195.425,A 0.000,B 0.000,C 90.000,E1 112.514} C_DIS
LIN {X 0.024,Y -686.419,Z 1195.424,A 0.000,B 0.000,C 90.000,E1 112.333} C_DIS
LIN {X -0.311,Y -685.150,Z 1195.424,A 0.000,B 0.000,C 90.000,E1 112.333} C_DIS
LIN {X 0.073,Y -681.768,Z 1195.424,A 0.000,B 0.000,C 90.000,E1 112.280} C_DIS
LIN {X -0.064,Y -677.999,Z 1195.424,A 0.000,B 0.000,C 90.000,E1 112.280} C_DIS
LIN {X -0.104,Y -607.636,Z 1195.424,A 0.000,B 0.000,C 90.000,E1 112.280} C_DIS
LIN {X -0.086,Y -601.965,Z 1195.422,A 0.000,B 0.000,C 90.000,E1 111.897} C_DIS
LIN {X 0.032,Y -593.153,Z 1195.418,A 0.000,B 0.000,C 90.000,E1 111.173} C_DIS
LIN {X 0.191,Y -584.473,Z 1195.414,A 0.000,B 0.000,C 90.000,E1 110.482} C_DIS
LIN {X 0.225,Y -575.732,Z 1195.410,A 0.000,B 0.000,C 90.000,E1 109.812} C_DIS
LIN {X 0.195,Y -574.789,Z 1195.410,A 0.000,B 0.000,C 90.000,E1 109.704} C_DIS
LIN {X 0.110,Y -573.358,Z 1195.409,A 0.000,B 0.000,C 90.000,E1 109.577} C_DIS
LIN {X 0.279,Y -571.870,Z 1195.408,A 0.000,B 0.000,C 90.000,E1 109.450} C_DIS
LIN {X 0.237,Y -571.841,Z 1195.408,A 0.000,B 0.000,C 90.000,E1 109.450} C_DIS
LIN {X -0.067,Y -571.347,Z 1195.407,A 0.000,B 0.000,C 90.000,E1 109.322} C_DIS
LIN {X -0.348,Y -571.158,Z 1195.407,A 0.000,B 0.000,C 90.000,E1 109.214} C_DIS
LIN {X 0.061,Y -571.423,Z 1195.406,A 0.000,B 0.000,C 90.000,E1 109.033} C_DIS
LIN {X 0.041,Y -573.126,Z 1195.403,A 0.000,B 0.000,C 90.000,E1 108.489} C_DIS
LIN {X 0.030,Y -575.008,Z 1195.400,A 0.000,B 0.000,C 90.000,E1 107.946} C_DIS
LIN {X -0.155,Y -576.939,Z 1195.395,A 0.000,B 0.000,C 90.000,E1 107.149} C_DIS
LIN {X -0.312,Y -577.830,Z 1195.392,A 0.000,B 0.000,C 90.000,E1 106.622} C_DIS
LIN {X -0.085,Y -578.715,Z 1195.388,A 0.000,B 0.000,C 90.000,E1 105.788} C_DIS
LIN {X -0.063,Y -579.164,Z 1195.385,A 0.000,B 0.000,C 90.000,E1 105.245} C_DIS
LIN {X 0.026,Y -578.715,Z 1195.380,A 0.000,B 0.000,C 90.000,E1 104.426} C_DIS
LIN {X 0.042,Y -578.110,Z 1195.377,A 0.000,B 0.000,C 90.000,E1 103.883} C_DIS
LIN {X 0.259,Y -577.618,Z 1195.376,A 0.000,B 0.000,C 90.000,E1 103.592} C_DIS
LIN {X 0.127,Y -576.187,Z 1195.373,A 0.000,B 0.000,C 90.000,E1 103.063} C_DIS
LIN {X -0.013,Y -574.358,Z 1195.370,A 0.000,B 0.000,C 90.000,E1 102.535} C_DIS
LIN {X -0.162,Y -571.769,Z 1195.367,A 0.000,B 0.000,C 90.000,E1 102.007} C_DIS
LIN {X -0.093,Y -569.357,Z 1195.364,A 0.000,B 0.000,C 90.000,E1 101.591} C_DIS
LIN {X -0.217,Y -563.574,Z 1195.360,A 0.000,B 0.000,C 90.000,E1 100.782} C_DIS
LIN {X -0.072,Y -561.704,Z 1195.358,A 0.000,B 0.000,C 90.000,E1 100.423} C_DIS
LIN {X 0.124,Y -560.425,Z 1195.355,A 0.000,B 0.000,C 90.000,E1 99.962} C_DIS
LIN {X -0.129,Y -560.396,Z 1195.355,A 0.000,B 0.000,C 90.000,E1 99.849} C_DIS
LIN {X 0.020,Y -559.942,Z 1195.353,A 0.000,B 0.000,C 90.000,E1 99.557} C_DIS
LIN {X -0.136,Y -559.568,Z 1195.352,A 0.000,B 0.000,C 90.000,E1 99.434} C_DIS
LIN {X -0.240,Y -559.539,Z 1195.350,A 0.000,B 0.000,C 90.000,E1 99.029} C_DIS
LIN {X 0.065,Y -559.363,Z 1195.349,A 0.000,B 0.000,C 90.000,E1 98.859} C_DIS
LIN {X 0.130,Y -559.654,Z 1195.344,A 0.000,B 0.000,C 90.000,E1 97.992} C_DIS
LIN {X -0.290,Y -560.669,Z 1195.337,A 0.000,B 0.000,C 90.000,E1 96.663} C_DIS
LIN {X -0.267,Y -561.717,Z 1195.329,A 0.000,B 0.000,C 90.000,E1 95.277} C_DIS
LIN {X -0.189,Y -562.838,Z 1195.320,A 0.000,B 0.000,C 90.000,E1 93.612} C_DIS
LIN {X -0.113,Y -563.982,Z 1195.311,A 0.000,B 0.000,C 90.000,E1 91.949} C_DIS
LIN {X -0.010,Y -565.229,Z 1195.302,A 0.000,B 0.000,C 90.000,E1 90.286} C_DIS
LIN {X 0.218,Y -566.621,Z 1195.291,A 0.000,B 0.000,C 90.000,E1 88.339} C_DIS
LIN {X -0.169,Y -567.815,Z 1195.282,A 0.000,B 0.000,C 90.000,E1 86.731} C_DIS
LIN {X 0.048,Y -569.064,Z 1195.273,A 0.000,B 0.000,C 90.000,E1 85.065} C_DIS
LIN {X 0.165,Y -570.029,Z 1195.265,A 0.000,B 0.000,C 90.000,E1 83.685} C_DIS
LIN {X -0.208,Y -571.032,Z 1195.257,A 0.000,B 0.000,C 90.000,E1 82.356} C_DIS
LIN {X -0.105,Y -571.799,Z 1195.251,A 0.000,B 0.000,C 90.000,E1 81.254} C_DIS
LIN {X -0.067,Y -572.974,Z 1195.241,A 0.000,B 0.000,C 90.000,E1 79.342} C_DIS
LIN {X -0.197,Y -573.802,Z 1195.233,A 0.000,B 0.000,C 90.000,E1 77.993} C_DIS
LIN {X 0.248,Y -574.489,Z 1195.226,A 0.000,B 0.000,C 90.000,E1 76.589} C_DIS
LIN {X 0.121,Y -575.456,Z 1195.215,A 0.000,B 0.000,C 90.000,E1 74.700} C_DIS
LIN {X -0.236,Y -575.895,Z 1195.211,A 0.000,B 0.000,C 90.000,E1 73.921} C_DIS
LIN {X -0.011,Y -576.878,Z 1195.200,A 0.000,B 0.000,C 90.000,E1 72.000} C_DIS
LIN {X 0.043,Y -577.884,Z 1195.191,A 0.000,B 0.000,C 90.000,E1 70.369} C_DIS
LIN {X -0.230,Y -579.025,Z 1195.182,A 0.000,B 0.000,C 90.000,E1 68.773} C_DIS
LIN {X -0.091,Y -580.656,Z 1195.172,A 0.000,B 0.000,C 90.000,E1 66.869} C_DIS
LIN {X -0.117,Y -581.776,Z 1195.166,A 0.000,B 0.000,C 90.000,E1 65.793} C_DIS
LIN {X -0.110,Y -583.771,Z 1195.154,A 0.000,B 0.000,C 90.000,E1 63.640} C_DIS
LIN {X -0.070,Y -585.416,Z 1195.145,A 0.000,B 0.000,C 90.000,E1 62.025} C_DIS
LIN {X -0.004,Y -587.001,Z 1195.136,A 0.000,B 0.000,C 90.000,E1 60.411} C_DIS
LIN {X -0.016,Y -588.176,Z 1195.128,A 0.000,B 0.000,C 90.000,E1 59.076} C_DIS
LIN {X 0.185,Y -589.472,Z 1195.119,A 0.000,B 0.000,C 90.000,E1 57.454} C_DIS
LIN {X -0.161,Y -590.295,Z 1195.113,A 0.000,B 0.000,C 90.000,E1 56.421} C_DIS
LIN {X 0.197,Y -591.280,Z 1195.106,A 0.000,B 0.000,C 90.000,E1 55.055} C_DIS
LIN {X -0.190,Y -592.487,Z 1195.097,A 0.000,B 0.000,C 90.000,E1 53.497} C_DIS
LIN {X -0.197,Y -593.587,Z 1195.088,A 0.000,B 0.000,C 90.000,E1 51.904} C_DIS
LIN {X -0.027,Y -594.353,Z 1195.081,A 0.000,B 0.000,C 90.000,E1 50.561} C_DIS
LIN {X -0.071,Y -595.220,Z 1195.072,A 0.000,B 0.000,C 90.000,E1 48.976} C_DIS
LIN {X 0.121,Y -595.617,Z 1195.065,A 0.000,B 0.000,C 90.000,E1 47.634} C_DIS
LIN {X 0.063,Y -595.835,Z 1195.059,A 0.000,B 0.000,C 90.000,E1 46.581} C_DIS
LIN {X 0.027,Y -595.900,Z 1195.053,A 0.000,B 0.000,C 90.000,E1 45.526} C_DIS
LIN {X -0.028,Y -595.806,Z 1195.047,A 0.000,B 0.000,C 90.000,E1 44.474} C_DIS
LIN {X -0.066,Y -595.482,Z 1195.041,A 0.000,B 0.000,C 90.000,E1 43.419} C_DIS
LIN {X -0.109,Y -595.293,Z 1195.038,A 0.000,B 0.000,C 90.000,E1 42.894} C_DIS
LIN {X -0.143,Y -594.637,Z 1195.032,A 0.000,B 0.000,C 90.000,E1 41.838} C_DIS
LIN {X 0.040,Y -593.671,Z 1195.025,A 0.000,B 0.000,C 90.000,E1 40.496} C_DIS
LIN {X -0.219,Y -593.071,Z 1195.021,A 0.000,B 0.000,C 90.000,E1 39.725} C_DIS
LIN {X -0.067,Y -591.802,Z 1195.013,A 0.000,B 0.000,C 90.000,E1 38.382} C_DIS
LIN {X 0.161,Y -590.141,Z 1195.006,A 0.000,B 0.000,C 90.000,E1 37.030} C_DIS
LIN {X -0.113,Y -588.121,Z 1194.998,A 0.000,B 0.000,C 90.000,E1 35.724} C_DIS
LIN {X -0.292,Y -585.559,Z 1194.991,A 0.000,B 0.000,C 90.000,E1 34.405} C_DIS
LIN {X -0.063,Y -583.513,Z 1194.987,A 0.000,B 0.000,C 90.000,E1 33.579} C_DIS
LIN {X 0.143,Y -581.252,Z 1194.982,A 0.000,B 0.000,C 90.000,E1 32.752} C_DIS
LIN {X 0.162,Y -579.592,Z 1194.979,A 0.000,B 0.000,C 90.000,E1 32.212} C_DIS
LIN {X 0.170,Y -577.740,Z 1194.976,A 0.000,B 0.000,C 90.000,E1 31.671} C_DIS
LIN {X 0.144,Y -573.483,Z 1194.970,A 0.000,B 0.000,C 90.000,E1 30.590} C_DIS
LIN {X -0.154,Y -569.001,Z 1194.965,A 0.000,B 0.000,C 90.000,E1 29.667} C_DIS
LIN {X 0.357,Y -566.951,Z 1194.963,A 0.000,B 0.000,C 90.000,E1 29.205} C_DIS
LIN {X -0.024,Y -561.791,Z 1194.957,A 0.000,B 0.000,C 90.000,E1 28.281} C_DIS
LIN {X -0.025,Y -557.663,Z 1194.953,A 0.000,B 0.000,C 90.000,E1 27.590} C_DIS
LIN {X -0.025,Y -551.491,Z 1194.948,A 0.000,B 0.000,C 90.000,E1 26.616} C_DIS
LIN {X -0.105,Y -546.578,Z 1194.944,A 0.000,B 0.000,C 90.000,E1 25.924} C_DIS
LIN {X 0.133,Y -542.337,Z 1194.941,A 0.000,B 0.000,C 90.000,E1 25.335} C_DIS
LIN {X 0.017,Y -536.644,Z 1194.937,A 0.000,B 0.000,C 90.000,E1 24.643} C_DIS
LIN {X 0.196,Y -529.452,Z 1194.932,A 0.000,B 0.000,C 90.000,E1 23.770} C_DIS
LIN {X 0.114,Y -524.260,Z 1194.929,A 0.000,B 0.000,C 90.000,E1 23.206} C_DIS
LIN {X 0.226,Y -514.967,Z 1194.924,A 0.000,B 0.000,C 90.000,E1 22.206} C_DIS
LIN {X -0.167,Y -505.449,Z 1194.918,A 0.000,B 0.000,C 90.000,E1 21.280} C_DIS
LIN {X 0.168,Y -494.259,Z 1194.912,A 0.000,B 0.000,C 90.000,E1 20.174} C_DIS
LIN {X 0.064,Y -485.542,Z 1194.908,A 0.000,B 0.000,C 90.000,E1 19.396} C_DIS
LIN {X 0.116,Y -476.869,Z 1194.903,A 0.000,B 0.000,C 90.000,E1 18.598} C_DIS
LIN {X 0.068,Y -469.429,Z 1194.900,A 0.000,B 0.000,C 90.000,E1 17.946} C_DIS
LIN {X 0.084,Y -448.775,Z 1194.889,A 0.000,B 0.000,C 90.000,E1 16.079} C_DIS
LIN {X 0.212,Y -428.438,Z 1194.878,A 0.000,B 0.000,C 90.000,E1 14.064} C_DIS
LIN {X 0.097,Y -414.416,Z 1194.870,A 0.000,B 0.000,C 90.000,E1 12.535} C_DIS
LIN {X -0.147,Y -403.502,Z 1194.862,A 0.000,B 0.000,C 90.000,E1 11.243} C_DIS
LIN {X -0.145,Y -398.378,Z 1194.859,A 0.000,B 0.000,C 90.000,E1 10.546} C_DIS
LIN {X -0.159,Y -396.058,Z 1194.857,A 0.000,B 0.000,C 90.000,E1 10.197} C_DIS
LIN {X 0.139,Y -393.786,Z 1194.854,A 0.000,B 0.000,C 90.000,E1 9.670} C_DIS
LIN {X -0.089,Y -393.641,Z 1194.854,A 0.000,B 0.000,C 90.000,E1 9.670} C_DIS
LIN {X -0.126,Y -393.622,Z 1194.854,A 0.000,B 0.000,C 90.000,E1 9.670} C_DIS
LIN {X -0.125,Y -393.230,Z 1194.852,A 0.000,B 0.000,C 90.000,E1 9.321} C_DIS
LIN {X -0.163,Y -393.238,Z 1194.852,A 0.000,B 0.000,C 90.000,E1 9.321} C_DIS
LIN {X 0.098,Y -394.326,Z 1194.849,A 0.000,B 0.000,C 90.000,E1 8.746} C_DIS
LIN {X -0.125,Y -397.292,Z 1194.845,A 0.000,B 0.000,C 90.000,E1 8.049} C_DIS
LIN {X 0.075,Y -402.331,Z 1194.840,A 0.000,B 0.000,C 90.000,E1 7.239} C_DIS
LIN {X -0.094,Y -406.940,Z 1194.838,A 0.000,B 0.000,C 90.000,E1 6.777} C_DIS
LIN {X 0.150,Y -415.013,Z 1194.834,A 0.000,B 0.000,C 90.000,E1 6.087} C_DIS
LIN {X 0.024,Y -429.471,Z 1194.828,A 0.000,B 0.000,C 90.000,E1 4.992} C_DIS
LIN {X -0.220,Y -439.034,Z 1194.824,A 0.000,B 0.000,C 90.000,E1 4.302} C_DIS
LIN {X 0.012,Y -451.863,Z 1194.818,A 0.000,B 0.000,C 90.000,E1 3.326} C_DIS
LIN {X -0.050,Y -466.166,Z 1194.813,A 0.000,B 0.000,C 90.000,E1 2.293} C_DIS
LIN {X -0.161,Y -473.882,Z 1194.809,A 0.000,B 0.000,C 90.000,E1 1.718} C_DIS
LIN {X 0.037,Y -481.459,Z 1194.806,A 0.000,B 0.000,C 90.000,E1 1.088} C_DIS
LIN {X -0.067,Y -485.701,Z 1194.804,A 0.000,B 0.000,C 90.000,E1 0.745} C_DIS
LIN {X -0.016,Y -491.497,Z 1194.801,A 0.000,B 0.000,C 90.000,E1 0.229} C_DIS
LIN {X 0.013,Y -497.464,Z 1194.798,A 0.000,B 0.000,C 90.000,E1 359.656} C_DIS
LIN {X 0.053,Y -504.115,Z 1194.794,A 0.000,B 0.000,C 90.000,E1 358.969} C_DIS
LIN {X 0.248,Y -510.451,Z 1194.790,A 0.000,B 0.000,C 90.000,E1 358.224} C_DIS
LIN {X -0.199,Y -516.556,Z 1194.786,A 0.000,B 0.000,C 90.000,E1 357.535} C_DIS
LIN {X 0.155,Y -523.111,Z 1194.781,A 0.000,B 0.000,C 90.000,E1 356.617} C_DIS
LIN {X 0.061,Y -527.150,Z 1194.778,A 0.000,B 0.000,C 90.000,E1 356.045} C_DIS
LIN {X -0.247,Y -531.676,Z 1194.774,A 0.000,B 0.000,C 90.000,E1 355.355} C_DIS
LIN {X -0.246,Y -535.060,Z 1194.771,A 0.000,B 0.000,C 90.000,E1 354.780} C_DIS
LIN {X 0.045,Y -538.764,Z 1194.767,A 0.000,B 0.000,C 90.000,E1 354.033} C_DIS
LIN {X -0.105,Y -542.177,Z 1194.763,A 0.000,B 0.000,C 90.000,E1 353.337} C_DIS
LIN {X -0.289,Y -545.274,Z 1194.759,A 0.000,B 0.000,C 90.000,E1 352.648} C_DIS
LIN {X -0.103,Y -548.629,Z 1194.754,A 0.000,B 0.000,C 90.000,E1 351.781} C_DIS
LIN {X 0.207,Y -551.654,Z 1194.750,A 0.000,B 0.000,C 90.000,E1 350.905} C_DIS
LIN {X 0.042,Y -555.225,Z 1194.743,A 0.000,B 0.000,C 90.000,E1 349.803} C_DIS
LIN {X 0.057,Y -559.151,Z 1194.736,A 0.000,B 0.000,C 90.000,E1 348.409} C_DIS
LIN {X 0.091,Y -561.956,Z 1194.729,A 0.000,B 0.000,C 90.000,E1 347.297} C_DIS
LIN {X -0.255,Y -564.538,Z 1194.723,A 0.000,B 0.000,C 90.000,E1 346.228} C_DIS
LIN {X 0.161,Y -567.560,Z 1194.716,A 0.000,B 0.000,C 90.000,E1 344.810} C_DIS
LIN {X 0.277,Y -569.245,Z 1194.711,A 0.000,B 0.000,C 90.000,E1 343.976} C_DIS
LIN {X 0.013,Y -572.393,Z 1194.702,A 0.000,B 0.000,C 90.000,E1 342.362} C_DIS
LIN {X -0.013,Y -574.317,Z 1194.696,A 0.000,B 0.000,C 90.000,E1 341.275} C_DIS
LIN {X -0.016,Y -575.977,Z 1194.690,A 0.000,B 0.000,C 90.000,E1 340.188} C_DIS
LIN {X 0.202,Y -577.393,Z 1194.684,A 0.000,B 0.000,C 90.000,E1 339.082} C_DIS
LIN {X 0.058,Y -578.240,Z 1194.679,A 0.000,B 0.000,C 90.000,E1 338.284} C_DIS
LIN {X -0.229,Y -579.050,Z 1194.673,A 0.000,B 0.000,C 90.000,E1 337.230} C_DIS
LIN {X -0.132,Y -579.312,Z 1194.669,A 0.000,B 0.000,C 90.000,E1 336.410} C_DIS
LIN {X -0.267,Y -579.234,Z 1194.664,A 0.000,B 0.000,C 90.000,E1 335.613} C_DIS
LIN {X -0.168,Y -578.853,Z 1194.660,A 0.000,B 0.000,C 90.000,E1 334.793} C_DIS
LIN {X 0.068,Y -578.391,Z 1194.657,A 0.000,B 0.000,C 90.000,E1 334.229} C_DIS
LIN {X 0.036,Y -577.782,Z 1194.654,A 0.000,B 0.000,C 90.000,E1 333.691} C_DIS
LIN {X 0.117,Y -576.522,Z 1194.649,A 0.000,B 0.000,C 90.000,E1 332.871} C_DIS
LIN {X -0.332,Y -574.848,Z 1194.645,A 0.000,B 0.000,C 90.000,E1 332.103} C_DIS
LIN {X -0.024,Y -572.883,Z 1194.640,A 0.000,B 0.000,C 90.000,E1 331.257} C_DIS
LIN {X -0.236,Y -570.561,Z 1194.636,A 0.000,B 0.000,C 90.000,E1 330.461} C_DIS
LIN {X 0.198,Y -568.640,Z 1194.633,A 0.000,B 0.000,C 90.000,E1 329.871} C_DIS
LIN {X 0.219,Y -566.990,Z 1194.630,A 0.000,B 0.000,C 90.000,E1 329.459} C_DIS
LIN {X -0.155,Y -564.279,Z 1194.627,A 0.000,B 0.000,C 90.000,E1 328.948} C_DIS
LIN {X -0.256,Y -561.369,Z 1194.624,A 0.000,B 0.000,C 90.000,E1 328.408} C_DIS
LIN {X 0.283,Y -556.922,Z 1194.621,A 0.000,B 0.000,C 90.000,E1 327.661} C_DIS
LIN {X 0.193,Y -550.991,Z 1194.616,A 0.000,B 0.000,C 90.000,E1 326.834} C_DIS
LIN {X 0.125,Y -547.800,Z 1194.614,A 0.000,B 0.000,C 90.000,E1 326.421} C_DIS
LIN {X 0.080,Y -542.042,Z 1194.610,A 0.000,B 0.000,C 90.000,E1 325.722} C_DIS
LIN {X -0.158,Y -534.864,Z 1194.605,A 0.000,B 0.000,C 90.000,E1 324.895} C_DIS
LIN {X -0.112,Y -527.406,Z 1194.600,A 0.000,B 0.000,C 90.000,E1 324.036} C_DIS
LIN {X -0.022,Y -522.590,Z 1194.597,A 0.000,B 0.000,C 90.000,E1 323.463} C_DIS
LIN {X 0.172,Y -519.594,Z 1194.595,A 0.000,B 0.000,C 90.000,E1 323.050} C_DIS
LIN {X -0.060,Y -516.721,Z 1194.592,A 0.000,B 0.000,C 90.000,E1 322.637} C_DIS
LIN {X 0.003,Y -514.590,Z 1194.590,A 0.000,B 0.000,C 90.000,E1 322.190} C_DIS
LIN {X 0.127,Y -514.034,Z 1194.589,A 0.000,B 0.000,C 90.000,E1 322.029} C_DIS
LIN {X -0.185,Y -512.556,Z 1194.586,A 0.000,B 0.000,C 90.000,E1 321.457} C_DIS
LIN {X -0.142,Y -512.125,Z 1194.583,A 0.000,B 0.000,C 90.000,E1 321.009} C_DIS
LIN {X -0.267,Y -511.946,Z 1194.580,A 0.000,B 0.000,C 90.000,E1 320.436} C_DIS
LIN {X -0.081,Y -513.340,Z 1194.565,A 0.000,B 0.000,C 90.000,E1 317.757} C_DIS
LIN {X -0.114,Y -514.039,Z 1194.559,A 0.000,B 0.000,C 90.000,E1 316.581} C_DIS
LIN {X -0.068,Y -515.175,Z 1194.547,A 0.000,B 0.000,C 90.000,E1 314.514} C_DIS
LIN {X 0.194,Y -516.026,Z 1194.539,A 0.000,B 0.000,C 90.000,E1 313.014} C_DIS
LIN {X -0.137,Y -517.483,Z 1194.526,A 0.000,B 0.000,C 90.000,E1 310.701} C_DIS
LIN {X 0.087,Y -518.759,Z 1194.515,A 0.000,B 0.000,C 90.000,E1 308.624} C_DIS
LIN {X 0.179,Y -519.384,Z 1194.508,A 0.000,B 0.000,C 90.000,E1 307.443} C_DIS
LIN {X -0.146,Y -520.251,Z 1194.498,A 0.000,B 0.000,C 90.000,E1 305.724} C_DIS
LIN {X 0.012,Y -520.924,Z 1194.490,A 0.000,B 0.000,C 90.000,E1 304.246} C_DIS
LIN {X -0.009,Y -521.835,Z 1194.481,A 0.000,B 0.000,C 90.000,E1 302.498} C_DIS
LIN {X -0.119,Y -522.404,Z 1194.473,A 0.000,B 0.000,C 90.000,E1 301.052} C_DIS
LIN {X 0.334,Y -522.700,Z 1194.468,A 0.000,B 0.000,C 90.000,E1 300.129} C_DIS
LIN {X 0.151,Y -522.962,Z 1194.460,A 0.000,B 0.000,C 90.000,E1 298.693} C_DIS
LIN {X -0.026,Y -523.195,Z 1194.451,A 0.000,B 0.000,C 90.000,E1 297.257} C_DIS
LIN {X 0.028,Y -523.392,Z 1194.443,A 0.000,B 0.000,C 90.000,E1 295.796} C_DIS
LIN {X 0.089,Y -523.418,Z 1194.435,A 0.000,B 0.000,C 90.000,E1 294.335} C_DIS
LIN {X -0.069,Y -523.320,Z 1194.427,A 0.000,B 0.000,C 90.000,E1 292.898} C_DIS
LIN {X -0.103,Y -523.273,Z 1194.416,A 0.000,B 0.000,C 90.000,E1 290.865} C_DIS
LIN {X 0.184,Y -523.063,Z 1194.406,A 0.000,B 0.000,C 90.000,E1 289.087} C_DIS
LIN {X -0.012,Y -522.826,Z 1194.401,A 0.000,B 0.000,C 90.000,E1 288.236} C_DIS
LIN {X -0.089,Y -521.822,Z 1194.390,A 0.000,B 0.000,C 90.000,E1 286.205} C_DIS
LIN {X 0.185,Y -521.079,Z 1194.384,A 0.000,B 0.000,C 90.000,E1 285.009} C_DIS
LIN {X -0.199,Y -520.043,Z 1194.375,A 0.000,B 0.000,C 90.000,E1 283.592} C_DIS
LIN {X -0.103,Y -518.842,Z 1194.366,A 0.000,B 0.000,C 90.000,E1 281.827} C_DIS
LIN {X -0.136,Y -517.964,Z 1194.358,A 0.000,B 0.000,C 90.000,E1 280.366} C_DIS
LIN {X 0.205,Y -516.848,Z 1194.346,A 0.000,B 0.000,C 90.000,E1 278.276} C_DIS
LIN {X -0.111,Y -515.935,Z 1194.336,A 0.000,B 0.000,C 90.000,E1 276.549} C_DIS
LIN {X 0.238,Y -515.162,Z 1194.330,A 0.000,B 0.000,C 90.000,E1 275.334} C_DIS
LIN {X -0.035,Y -514.498,Z 1194.323,A 0.000,B 0.000,C 90.000,E1 274.188} C_DIS
LIN {X -0.138,Y -513.100,Z 1194.309,A 0.000,B 0.000,C 90.000,E1 271.547} C_DIS
LIN {X -0.095,Y -512.252,Z 1194.299,A 0.000,B 0.000,C 90.000,E1 269.771} C_DIS
LIN {X 0.093,Y -511.668,Z 1194.292,A 0.000,B 0.000,C 90.000,E1 268.568} C_DIS
LIN {X -0.047,Y -510.129,Z 1194.279,A 0.000,B 0.000,C 90.000,E1 266.216} C_DIS
LIN {X 0.158,Y -509.271,Z 1194.272,A 0.000,B 0.000,C 90.000,E1 265.008} C_DIS
LIN {X -0.262,Y -507.786,Z 1194.264,A 0.000,B 0.000,C 90.000,E1 263.571} C_DIS
LIN {X 0.235,Y -505.950,Z 1194.253,A 0.000,B 0.000,C 90.000,E1 261.432} C_DIS
LIN {X -0.237,Y -504.272,Z 1194.241,A 0.000,B 0.000,C 90.000,E1 259.398} C_DIS
LIN {X -0.058,Y -502.532,Z 1194.229,A 0.000,B 0.000,C 90.000,E1 257.285} C_DIS
LIN {X 0.071,Y -500.782,Z 1194.218,A 0.000,B 0.000,C 90.000,E1 255.172} C_DIS
LIN {X -0.123,Y -498.737,Z 1194.203,A 0.000,B 0.000,C 90.000,E1 252.489} C_DIS
LIN {X -0.044,Y -497.929,Z 1194.196,A 0.000,B 0.000,C 90.000,E1 251.275} C_DIS
LIN {X 0.020,Y -496.146,Z 1194.184,A 0.000,B 0.000,C 90.000,E1 249.156} C_DIS
LIN {X -0.126,Y -494.482,Z 1194.174,A 0.000,B 0.000,C 90.000,E1 247.358} C_DIS
LIN {X 0.257,Y -493.280,Z 1194.167,A 0.000,B 0.000,C 90.000,E1 246.102} C_DIS
LIN {X 0.214,Y -491.786,Z 1194.159,A 0.000,B 0.000,C 90.000,E1 244.588} C_DIS
LIN {X -0.059,Y -489.651,Z 1194.149,A 0.000,B 0.000,C 90.000,E1 242.794} C_DIS
LIN {X -0.216,Y -488.556,Z 1194.144,A 0.000,B 0.000,C 90.000,E1 241.897} C_DIS
LIN {X 0.084,Y -486.634,Z 1194.135,A 0.000,B 0.000,C 90.000,E1 240.333} C_DIS
LIN {X -0.270,Y -484.296,Z 1194.125,A 0.000,B 0.000,C 90.000,E1 238.535} C_DIS
LIN {X 0.244,Y -481.928,Z 1194.115,A 0.000,B 0.000,C 90.000,E1 236.628} C_DIS
LIN {X 0.103,Y -479.137,Z 1194.103,A 0.000,B 0.000,C 90.000,E1 234.482} C_DIS
LIN {X 0.175,Y -477.227,Z 1194.094,A 0.000,B 0.000,C 90.000,E1 232.924} C_DIS
LIN {X 0.162,Y -474.174,Z 1194.080,A 0.000,B 0.000,C 90.000,E1 230.436} C_DIS
LIN {X -0.310,Y -472.296,Z 1194.072,A 0.000,B 0.000,C 90.000,E1 228.933} C_DIS
LIN {X -0.077,Y -469.941,Z 1194.061,A 0.000,B 0.000,C 90.000,E1 227.025} C_DIS
LIN {X -0.038,Y -466.754,Z 1194.046,A 0.000,B 0.000,C 90.000,E1 224.190} C_DIS
LIN {X -0.147,Y -464.593,Z 1194.031,A 0.000,B 0.000,C 90.000,E1 221.676} C_DIS
LIN {X 0.015,Y -463.614,Z 1194.010,A 0.000,B 0.000,C 90.000,E1 217.855} C_DIS
LIN {X -0.202,Y -463.724,Z 1194.002,A 0.000,B 0.000,C 90.000,E1 216.297} C_DIS
LIN {X 0.249,Y -464.053,Z 1193.987,A 0.000,B 0.000,C 90.000,E1 213.706} C_DIS
LIN {X -0.150,Y -466.208,Z 1193.970,A 0.000,B 0.000,C 90.000,E1 210.590} C_DIS
LIN {X 0.279,Y -469.345,Z 1193.952,A 0.000,B 0.000,C 90.000,E1 207.385} C_DIS
LIN {X 0.006,Y -471.100,Z 1193.944,A 0.000,B 0.000,C 90.000,E1 205.848} C_DIS
LIN {X 0.093,Y -478.055,Z 1193.918,A 0.000,B 0.000,C 90.000,E1 201.153} C_DIS
LIN {X -0.010,Y -485.282,Z 1193.899,A 0.000,B 0.000,C 90.000,E1 197.764} C_DIS
LIN {X 0.102,Y -490.873,Z 1193.887,A 0.000,B 0.000,C 90.000,E1 195.607} C_DIS
LIN {X 0.105,Y -496.982,Z 1193.875,A 0.000,B 0.000,C 90.000,E1 193.480} C_DIS
LIN {X 0.162,Y -503.447,Z 1193.863,A 0.000,B 0.000,C 90.000,E1 191.366} C_DIS
LIN {X 0.240,Y -511.191,Z 1193.850,A 0.000,B 0.000,C 90.000,E1 188.973} C_DIS
LIN {X -0.072,Y -516.167,Z 1193.842,A 0.000,B 0.000,C 90.000,E1 187.530} C_DIS
LIN {X 0.227,Y -521.014,Z 1193.834,A 0.000,B 0.000,C 90.000,E1 186.030} C_DIS
LIN {X 0.047,Y -527.714,Z 1193.822,A 0.000,B 0.000,C 90.000,E1 184.012} C_DIS
LIN {X -0.037,Y -531.517,Z 1193.816,A 0.000,B 0.000,C 90.000,E1 182.865} C_DIS
LIN {X -0.070,Y -536.273,Z 1193.808,A 0.000,B 0.000,C 90.000,E1 181.432} C_DIS
LIN {X 0.016,Y -542.926,Z 1193.797,A 0.000,B 0.000,C 90.000,E1 179.427} C_DIS
LIN {X 0.140,Y -546.640,Z 1193.791,A 0.000,B 0.000,C 90.000,E1 178.282} C_DIS
LIN {X -0.217,Y -550.386,Z 1193.784,A 0.000,B 0.000,C 90.000,E1 177.192} C_DIS
LIN {X -0.027,Y -553.184,Z 1193.780,A 0.000,B 0.000,C 90.000,E1 176.331} C_DIS
LIN {X -0.111,Y -558.524,Z 1193.770,A 0.000,B 0.000,C 90.000,E1 174.666} C_DIS
LIN {X -0.116,Y -562.957,Z 1193.763,A 0.000,B 0.000,C 90.000,E1 173.280} C_DIS
LIN {X 0.132,Y -568.172,Z 1193.753,A 0.000,B 0.000,C 90.000,E1 171.602} C_DIS
LIN {X -0.077,Y -573.299,Z 1193.744,A 0.000,B 0.000,C 90.000,E1 169.982} C_DIS
LIN {X 0.163,Y -576.661,Z 1193.738,A 0.000,B 0.000,C 90.000,E1 168.870} C_DIS
LIN {X -0.225,Y -581.808,Z 1193.729,A 0.000,B 0.000,C 90.000,E1 167.285} C_DIS
LIN {X 0.054,Y -586.859,Z 1193.720,A 0.000,B 0.000,C 90.000,E1 165.644} C_DIS
LIN {X -0.192,Y -589.417,Z 1193.716,A 0.000,B 0.000,C 90.000,E1 164.866} C_DIS
LIN {X 0.245,Y -595.326,Z 1193.706,A 0.000,B 0.000,C 90.000,E1 162.960} C_DIS
LIN {X -0.039,Y -600.426,Z 1193.697,A 0.000,B 0.000,C 90.000,E1 161.402} C_DIS
LIN {X -0.111,Y -606.212,Z 1193.687,A 0.000,B 0.000,C 90.000,E1 159.571} C_DIS
LIN {X 0.227,Y -611.138,Z 1193.678,A 0.000,B 0.000,C 90.000,E1 157.975} C_DIS
LIN {X 0.091,Y -616.041,Z 1193.669,A 0.000,B 0.000,C 90.000,E1 156.433} C_DIS
LIN {X -0.002,Y -620.003,Z 1193.662,A 0.000,B 0.000,C 90.000,E1 155.153} C_DIS
LIN {X -0.287,Y -623.089,Z 1193.656,A 0.000,B 0.000,C 90.000,E1 154.152} C_DIS
LIN {X -0.253,Y -626.756,Z 1193.649,A 0.000,B 0.000,C 90.000,E1 152.871} C_DIS
LIN {X 0.136,Y -630.365,Z 1193.642,A 0.000,B 0.000,C 90.000,E1 151.563} C_DIS
LIN {X -0.236,Y -634.484,Z 1193.634,A 0.000,B 0.000,C 90.000,E1 150.078} C_DIS
LIN {X -0.314,Y -637.104,Z 1193.628,A 0.000,B 0.000,C 90.000,E1 149.076} C_DIS
LIN {X 0.026,Y -640.214,Z 1193.621,A 0.000,B 0.000,C 90.000,E1 147.788} C_DIS
LIN {X 0.021,Y -642.576,Z 1193.616,A 0.000,B 0.000,C 90.000,E1 146.786} C_DIS
LIN {X -0.139,Y -644.774,Z 1193.610,A 0.000,B 0.000,C 90.000,E1 145.801} C_DIS
LIN {X -0.211,Y -647.395,Z 1193.603,A 0.000,B 0.000,C 90.000,E1 144.562} C_DIS
LIN {X 0.127,Y -649.784,Z 1193.596,A 0.000,B 0.000,C 90.000,E1 143.290} C_DIS
LIN {X -0.084,Y -652.608,Z 1193.588,A 0.000,B 0.000,C 90.000,E1 141.823} C_DIS
LIN {X 0.221,Y -655.911,Z 1193.578,A 0.000,B 0.000,C 90.000,E1 140.070} C_DIS
LIN {X 0.057,Y -658.939,Z 1193.570,A 0.000,B 0.000,C 90.000,E1 138.609} C_DIS
LIN {X -0.022,Y -661.621,Z 1193.563,A 0.000,B 0.000,C 90.000,E1 137.391} C_DIS
LIN {X 0.378,Y -664.716,Z 1193.555,A 0.000,B 0.000,C 90.000,E1 135.891} C_DIS
LIN {X 0.379,Y -669.581,Z 1193.543,A 0.000,B 0.000,C 90.000,E1 133.704} C_DIS
LIN {X 0.005,Y -673.652,Z 1193.534,A 0.000,B 0.000,C 90.000,E1 132.043} C_DIS
LIN {X -0.235,Y -677.720,Z 1193.524,A 0.000,B 0.000,C 90.000,E1 130.378} C_DIS
LIN {X 0.078,Y -680.691,Z 1193.518,A 0.000,B 0.000,C 90.000,E1 129.152} C_DIS
LIN {X 0.311,Y -683.020,Z 1193.512,A 0.000,B 0.000,C 90.000,E1 128.177} C_DIS
LIN {X -0.200,Y -686.640,Z 1193.504,A 0.000,B 0.000,C 90.000,E1 126.790} C_DIS
LIN {X -0.139,Y -689.582,Z 1193.498,A 0.000,B 0.000,C 90.000,E1 125.598} C_DIS
LIN {X 0.333,Y -691.788,Z 1193.492,A 0.000,B 0.000,C 90.000,E1 124.612} C_DIS
LIN {X 0.122,Y -695.071,Z 1193.485,A 0.000,B 0.000,C 90.000,E1 123.214} C_DIS
LIN {X -0.075,Y -697.578,Z 1193.478,A 0.000,B 0.000,C 90.000,E1 122.054} C_DIS
LIN {X -0.262,Y -699.505,Z 1193.473,A 0.000,B 0.000,C 90.000,E1 121.131} C_DIS
LIN {X 0.204,Y -701.734,Z 1193.466,A 0.000,B 0.000,C 90.000,E1 119.922} C_DIS
LIN {X 0.353,Y -703.686,Z 1193.460,A 0.000,B 0.000,C 90.000,E1 118.743} C_DIS
LIN {X -0.086,Y -705.078,Z 1193.455,A 0.000,B 0.000,C 90.000,E1 117.847} C_DIS
LIN {X 0.157,Y -705.874,Z 1193.451,A 0.000,B 0.000,C 90.000,E1 117.129} C_DIS
LIN {X 0.088,Y -706.384,Z 1193.447,A 0.000,B 0.000,C 90.000,E1 116.437} C_DIS
LIN {X 0.336,Y -706.719,Z 1193.443,A 0.000,B 0.000,C 90.000,E1 115.720} C_DIS
LIN {X 0.279,Y -706.704,Z 1193.439,A 0.000,B 0.000,C 90.000,E1 115.027} C_DIS
LIN {X -0.070,Y -706.469,Z 1193.437,A 0.000,B 0.000,C 90.000,E1 114.591} C_DIS
LIN {X -0.130,Y -705.636,Z 1193.434,A 0.000,B 0.000,C 90.000,E1 114.131} C_DIS
LIN {X -0.127,Y -705.117,Z 1193.433,A 0.000,B 0.000,C 90.000,E1 113.898} C_DIS
LIN {X -0.339,Y -702.367,Z 1193.430,A 0.000,B 0.000,C 90.000,E1 113.334} C_DIS
LIN {X -0.199,Y -701.535,Z 1193.429,A 0.000,B 0.000,C 90.000,E1 113.206} C_DIS
LIN {X 0.074,Y -698.975,Z 1193.428,A 0.000,B 0.000,C 90.000,E1 112.950} C_DIS
LIN {X 0.242,Y -696.360,Z 1193.426,A 0.000,B 0.000,C 90.000,E1 112.717} C_DIS
LIN {X -0.163,Y -694.917,Z 1193.426,A 0.000,B 0.000,C 90.000,E1 112.642} C_DIS
LIN {X 0.073,Y -692.522,Z 1193.425,A 0.000,B 0.000,C 90.000,E1 112.514} C_DIS
LIN {X -0.012,Y -686.386,Z 1193.424,A 0.000,B 0.000,C 90.000,E1 112.333} C_DIS
LIN {X 0.249,Y -684.885,Z 1193.424,A 0.000,B 0.000,C 90.000,E1 112.280} C_DIS
LIN {X -0.122,Y -677.867,Z 1193.424,A 0.000,B 0.000,C 90.000,E1 112.280} C_DIS
LIN {X -0.156,Y -607.341,Z 1193.424,A 0.000,B 0.000,C 90.000,E1 112.280} C_DIS
LIN {X 0.235,Y -602.129,Z 1193.422,A 0.000,B 0.000,C 90.000,E1 111.897} C_DIS
LIN {X 0.045,Y -592.077,Z 1193.417,A 0.000,B 0.000,C 90.000,E1 111.099} C_DIS
LIN {X 0.033,Y -583.387,Z 1193.414,A 0.000,B 0.000,C 90.000,E1 110.429} C_DIS
LIN {X -0.329,Y -571.752,Z 1193.409,A 0.000,B 0.000,C 90.000,E1 109.577} C_DIS
LIN {X -0.182,Y -569.530,Z 1193.408,A 0.000,B 0.000,C 90.000,E1 109.396} C_DIS
LIN {X -0.002,Y -568.126,Z 1193.407,A 0.000,B 0.000,C 90.000,E1 109.214} C_DIS
LIN {X -0.098,Y -566.591,Z 1193.406,A 0.000,B 0.000,C 90.000,E1 109.087} C_DIS
LIN {X -0.140,Y -566.570,Z 1193.406,A 0.000,B 0.000,C 90.000,E1 109.087} C_DIS
LIN {X -0.195,Y -566.768,Z 1193.405,A 0.000,B 0.000,C 90.000,E1 108.960} C_DIS
LIN {X -0.047,Y -567.445,Z 1193.404,A 0.000,B 0.000,C 90.000,E1 108.671} C_DIS
